// TwinCAT 3 PLC project PLC_CRIX_MOT
// Title: lcls-plc-crix-motion
// Company: SLAC
// ProjectVersion: 0.0.0
// ProgramVersion: 3.1.4023.0
// libraries:
//   LCLS General, * (SLAC)
//   lcls-twincat-motion, * (SLAC)
//   PMPS, * (SLAC - LCLS)
//   Tc2_MC2, * (Beckhoff Automation GmbH)
//   Tc2_Standard, * (Beckhoff Automation GmbH)
//   Tc2_System, * (Beckhoff Automation GmbH)
//   Tc3_EventLogger, * (Beckhoff Automation GmbH)
//   Tc3_Module, * (Beckhoff Automation GmbH)
// project tree:
//   DUTs/Assemblies/ ENUM_DiagPaddle.TcDUT (not stored), ENUM_DPX.TcDUT (not stored), ENUM_DPY.TcDUT (not stored), ENUM_DPZ.TcDUT (not stored), E_DPaddle_States.TcDUT (not stored), ST_DiagPaddleOutputs.TcDUT (not stored)
//   DUTs/EPS/ ST_BFSAssemblyState.TcDUT (not stored), ST_EPSLimits.TcDUT, ST_Queue.TcDUT (not stored)
//   GVLs/ GVL.TcGVL (not stored), GVL_DiagnosticPaddle.TcGVL (not stored), GVL_FiberLite.TcGVL, GVL_Illumination.TcGVL (not stored), GVL_MotorEPS.TcGVL, GVL_PMPS.TcGVL (not stored), GVL_PointDetector.TcGVL (not stored), GVL_Questar.TcGVL (not stored), GVL_SampleDelivery.TcGVL (not stored), Main.TcGVL
//   / PlcTask.TcTTO (not stored)
//   POUs/Assemblies/ FB_DPX.TcPOU (not stored), PRG_FZP.TcPOU, PRG_Camera.TcPOU (not stored), PRG_CryoPump.TcPOU, PRG_Cryopumps.TcPOU (not stored), PRG_CryoStat.TcPOU (not stored), PRG_DiagnosticPaddle.TcPOU (not stored), PRG_DiagnosticPaddleMotors.TcPOU (not stored), PRG_FiberLite.TcPOU, PRG_Illumination.TcPOU (not stored), PRG_InjectorMotors.TcPOU, PRG_PointDetectorMotors.TcPOU (not stored), PRG_ObjectivesMotors.TcPOU (not stored), PRG_QuestarMotors.TcPOU (not stored), PRG_RCC.TcPOU (not stored), PRG_RCI.TcPOU (not stored), PRG_VLS.TcPOU, PRG_SL2K2_SCATTER.TcPOU (not stored)
//   POUs/EPS/ FB_AdjacentStates.TcPOU (not stored), FB_AssemblyPositionStateManager.TcPOU (not stored), FB_BFS.TcPOU (not stored), FB_Queue.TcPOU (not stored), PRG_BFS.TcPOU (not stored), PRG_QueueTest.TcPOU (not stored), PRG_Test_AdjacentStates.TcPOU (not stored)
//   POUs/EPS/InjectorMotorEPSLimits/ FB_CheckEPS.TcPOU, F_InRange.TcPOU, FB_RestTimer.TcPOU, PRG_DPL_X_EPS.TcPOU, PRG_DPL_Y_EPS.TcPOU, PRG_DPL_Z_EPS.TcPOU, PRG_EPS.TcPOU, PRG_OBJ_X_EPS.TcPOU, PRG_RCC_Y_EPS.TcPOU, PRG_RCC_Z_EPS.TcPOU, PRG_SDS_RX_EPS.TcPOU, PRG_SDS_Y_EPS.TcPOU, PRG_SDS_ZENCODER_EPS.TcPOU
//   POUs/ FB_RCI_Analog_Input.TcPOU (not stored), FB_RCI_Analog_Output.TcPOU (not stored), PRG_Main.TcPOU, PRG_PMPS.TcPOU (not stored)
//   POUs/temp/ FB_SLITS.TcPOU (not stored), FB_SLITS_POWER.TcPOU (not stored), FB_SLITS_SCATTER.TcPOU (not stored)
// real-time tasks:
//   TASK PlcTask: cycle T#10ms, priority 20, ADS port 350
// motion (NC):
//   TASK NC-Task 1 SAF: cycle T#2ms, priority 4, ADS port 501
//   TASK NC-Task 1 SVB: cycle T#10ms, priority 8, ADS port 511
//   AXIS Cryo X (id 22)
//     Dynamic: AccelerationMaximum=1, DecelerationMaximum=1, Acceleration=1, Deceleration=1
//     Velo: Maximum=1.7
//     OtherSettings: AllowMotionCmdToSlave=true
//     encoder EncType=29
//       EncPara: ScaleFactorNumerator=5e-05, Offset=-31.22, MaxCount=#xffffffff, ReferenceSystem=1
//         Inc: RefSoftSyncMask=#x0000ffff
//     drive DrvType=24
//       DrvPara: Inverse=true
//         Analog: VeloReferenz=2, ScaleFactorActTorque=0.1
//         TimeComp: TaskDelayCycles=1
//     controller CtrType=2
//       CtrPara: PriorControlFactor=1
//         PosDiffControl: Range=0.5
//         PID: PosExtKp=1, DeadBandPosition=0.1
//         Observer: BandWidth=20
//   AXIS Cryo Y (id 23)
//     Dynamic: AccelerationMaximum=1, DecelerationMaximum=1, Acceleration=1, Deceleration=1
//     Velo: Maximum=1.4
//     OtherSettings: AllowMotionCmdToSlave=true
//     encoder EncType=29
//       EncPara: ScaleFactorNumerator=5e-05, Offset=-215.0149, MaxCount=#xffffffff
//         Inc: RefSoftSyncMask=#x0000ffff
//     drive DrvType=24
//       Analog: VeloReferenz=1.667, ScaleFactorActTorque=0.1
//       TimeComp: TaskDelayCycles=1
//     controller CtrType=2
//       CtrPara: PriorControlFactor=1
//         PosDiffControl: Range=0.5
//         PID: PosExtKp=1, DeadBandPosition=0.01
//         Observer: BandWidth=20
//   AXIS Cryo Z (id 24)
//     Dynamic: AccelerationMaximum=1, DecelerationMaximum=1, Acceleration=1, Deceleration=1
//     Velo: Maximum=1.7
//     OtherSettings: AllowMotionCmdToSlave=true
//     encoder EncType=29
//       EncPara: ScaleFactorNumerator=5e-05, Offset=-922337203685459, Inverse=true, MaxCount=#xffffffff, ReferenceSystem=1
//         Inc: RefSoftSyncMask=#x0000ffff
//     drive DrvType=24
//       DrvPara: Inverse=true
//         Analog: VeloReferenz=2, ScaleFactorActTorque=0.1
//         TimeComp: TaskDelayCycles=1
//     controller CtrType=2
//       CtrPara: PriorControlFactor=1
//         PosDiffControl: Range=0.5
//         PID: PosExtKp=1, DeadBandPosition=0.1
//         Observer: BandWidth=20
//   AXIS Cryo rY (id 25)
//   AXIS RCI X (id 26)
//     Dynamic: AccelerationMaximum=10, DecelerationMaximum=10, Acceleration=2, Deceleration=2
//     Velo: Maximum=0.4
//     OtherSettings: AllowMotionCmdToSlave=true
//     encoder EncType=29
//       EncPara: ScaleFactorNumerator=5e-05, Offset=-922337203685433, Inverse=true, MaxCount=#xffffffff, ReferenceSystem=1
//         Inc: RefSoftSyncMask=#x0000ffff
//     drive DrvType=24
//       Analog: VeloReferenz=2.667, ScaleFactorActTorque=0.1
//       TimeComp: TaskDelayCycles=1
//     controller CtrType=2
//       CtrPara: PriorControlFactor=1
//         PosDiffControl: Range=0.3
//         PID: PosExtKp=1, DeadBandPosition=0.1
//         Observer: BandWidth=20
//   AXIS RCI Y (id 27)
//     Dynamic: AccelerationMaximum=10, DecelerationMaximum=10, Acceleration=2, Deceleration=2
//     Velo: Maximum=1.7
//     OtherSettings: AllowMotionCmdToSlave=true
//     encoder EncType=29
//       EncPara: ScaleFactorNumerator=5e-05, Offset=-32.4565, MaxCount=#xffffffff, ReferenceSystem=1
//         Inc: RefSoftSyncMask=#x0000ffff
//     drive DrvType=24
//       Analog: VeloReferenz=2, ScaleFactorActTorque=0.1
//       TimeComp: TaskDelayCycles=1
//     controller CtrType=2
//       CtrPara: PriorControlFactor=1
//         PosDiffControl: Range=0.3
//         PID: DeadBandPosition=0.1
//         Observer: BandWidth=20
//   AXIS RCI Z (id 28)
//     Dynamic: AccelerationMaximum=10, DecelerationMaximum=10, Acceleration=2, Deceleration=2
//     Velo: Maximum=1.7
//     OtherSettings: AllowMotionCmdToSlave=true
//     encoder EncType=29
//       EncPara: ScaleFactorNumerator=5e-05, Offset=-922337203685442, Inverse=true, MaxCount=#xffffffff, ReferenceSystem=1
//         Inc: RefSoftSyncMask=#x0000ffff
//     drive DrvType=24
//       Analog: VeloReferenz=2, ScaleFactorActTorque=0.1
//       TimeComp: TaskDelayCycles=1
//     controller CtrType=2
//       CtrPara: PriorControlFactor=1
//         PosDiffControl: Range=0.3
//         PID: DeadBandPosition=0.1
//         Observer: BandWidth=20
//   AXIS RCI RX (id 29)
//     Dynamic: AccelerationMaximum=10, DecelerationMaximum=10, Acceleration=2, Deceleration=2
//     Velo: Maximum=2
//     OtherSettings: AllowMotionCmdToSlave=true
//     encoder EncType=4
//       EncPara: ScaleFactorNumerator=0.000234375, MaxCount=#x0000ffff
//         Inc: RefSoftSyncMask=#x0000ffff
//     drive DrvType=24
//       Analog: VeloReferenz=30, ScaleFactorActTorque=0.1
//       TimeComp: TaskDelayCycles=1
//     controller CtrType=2
//       CtrPara: PriorControlFactor=1
//         PosDiffControl: Range=0.3
//         PID: DeadBandPosition=0.5
//         Observer: BandWidth=20
//   AXIS FZP Y (id 30)
//     Dynamic: AccelerationMaximum=10, DecelerationMaximum=10, Acceleration=1, Deceleration=1
//     Velo: Maximum=2
//     OtherSettings: AllowMotionCmdToSlave=true
//     encoder EncType=29
//       EncPara: ScaleFactorNumerator=0.000244, Offset=-15658.9921, MaxCount=#xffffffff
//         Inc: RefSoftSyncMask=#x0000ffff
//     drive DrvType=24
//       DrvPara: Inverse=true
//         Analog: VeloReferenz=15, ScaleFactorActTorque=0.1
//         TimeComp: TaskDelayCycles=1
//     controller CtrType=2
//       CtrPara: PriorControlFactor=1
//         PosDiffControl: Range=0.5
//         PID: DeadBandPosition=0.01
//         Observer: BandWidth=20
//   AXIS FZP X (id 31)
//     Dynamic: AccelerationMaximum=10, DecelerationMaximum=10, Acceleration=1, Deceleration=1
//     Velo: Maximum=0.5
//     OtherSettings: AllowMotionCmdToSlave=true
//     encoder EncType=29
//       EncPara: ScaleFactorNumerator=0.000244, Offset=-16005.009, MaxCount=#xffffffff, ReferenceSystem=1
//         Inc: RefSoftSyncMask=#x0000ffff
//     drive DrvType=24
//       Analog: VeloReferenz=8, ScaleFactorActTorque=0.1
//       TimeComp: TaskDelayCycles=1
//     controller CtrType=2
//       CtrPara: PriorControlFactor=1
//         PosDiffControl: Range=0.5
//         PID: PosExtKp=1, DeadBandPosition=0.01
//         Observer: BandWidth=20
//   AXIS FZP Z (id 32)
//     Dynamic: AccelerationMaximum=10, DecelerationMaximum=10, Acceleration=1, Deceleration=1
//     Velo: Maximum=2
//     PositionAreaControl: Enable=false
//     OtherSettings: AllowMotionCmdToSlave=true
//     encoder EncType=29
//       EncPara: Offset=-1.0099, MaxCount=#xffffffff
//         Inc: RefSoftSyncMask=#x0000ffff
//     drive DrvType=24
//       Analog: VeloReferenz=15, ScaleFactorActTorque=0.1
//       TimeComp: TaskDelayCycles=1
//     controller CtrType=2
//       CtrPara: PriorControlFactor=1
//         PosDiffControl: Range=0.5
//         PID: DeadBandPosition=0.01
//         Observer: BandWidth=20
//   AXIS Camera X (id 33)
//   AXIS Camera Y (id 34)
//   AXIS M37-X (id 37)
//   AXIS M38-Y (id 38)
//   AXIS M39-Z (id 39)
//   AXIS M40-VLS-Slit-Top (id 40)
//     Dynamic: AccelerationMaximum=10, DecelerationMaximum=10, Acceleration=4.49102, Deceleration=4.49102, Jerk=20.1692
//     Velo: RefSearch=0.1, RefSync=0.1, SlowManual=0.5, FastManual=1, Maximum=1
//     OtherSettings: AllowMotionCmdToSlave=true, PulseDistancePos=1, PulseDistanceNeg=1
//     encoder EncType=4
//       EncPara: ScaleFactorNumerator=3.90625e-05, MaxCount=#x0000ffff
//         SoftEndMinControl: Enable=true
//         SoftEndMaxControl: Enable=true, Range=19
//         Inc: RefSoftSyncMask=#x0000ffff
//     drive DrvType=24
//       Analog: VeloReferenz=5, ScaleFactorActTorque=0.1
//       TimeComp: TaskDelayCycles=1
//     controller CtrType=2
//       CtrPara: PriorControlFactor=1
//         PosDiffControl: Range=0.1
//         PID: DeadBandPosition=0.1
//         Observer: BandWidth=20
//   AXIS M41-VLS-Slit-Bottom (id 41)
//     Dynamic: AccelerationMaximum=10, DecelerationMaximum=10, Acceleration=4.49102, Deceleration=4.49102, Jerk=20.1692
//     Velo: RefSearch=0.1, RefSync=0.1, SlowManual=0.5, FastManual=1, Maximum=1
//     OtherSettings: AllowMotionCmdToSlave=true, PulseDistancePos=1, PulseDistanceNeg=1
//     encoder EncType=4
//       EncPara: ScaleFactorNumerator=3.90625e-05, MaxCount=#x0000ffff
//         SoftEndMinControl: Enable=true
//         SoftEndMaxControl: Enable=true, Range=24.5
//         Inc: RefSoftSyncMask=#x0000ffff
//     drive DrvType=24
//       Analog: VeloReferenz=5, ScaleFactorActTorque=0.1
//       TimeComp: TaskDelayCycles=1
//     controller CtrType=2
//       CtrPara: PriorControlFactor=1
//         PosDiffControl: Range=0.1
//         PID: DeadBandPosition=0.1
//         Observer: BandWidth=20
//   AXIS M42-VLS-Slit-Right (id 42)
//     Dynamic: AccelerationMaximum=10, DecelerationMaximum=10, Acceleration=4.49102, Deceleration=4.49102, Jerk=20.1692
//     Velo: RefSearch=0.1, RefSync=0.1, SlowManual=0.5, FastManual=1, Maximum=1
//     OtherSettings: AllowMotionCmdToSlave=true, PulseDistancePos=1, PulseDistanceNeg=1
//     encoder EncType=4
//       EncPara: ScaleFactorNumerator=3.90625e-05, MaxCount=#x0000ffff
//         SoftEndMinControl: Enable=true
//         SoftEndMaxControl: Enable=true, Range=48.1
//         Inc: RefSoftSyncMask=#x0000ffff
//     drive DrvType=24
//       Analog: VeloReferenz=5, ScaleFactorActTorque=0.1
//       TimeComp: TaskDelayCycles=1
//     controller CtrType=2
//       CtrPara: PriorControlFactor=1
//         PosDiffControl: Range=0.1
//         PID: DeadBandPosition=0.1
//         Observer: BandWidth=20
//   AXIS M43-VLS-Slit-Left (id 43)
//     Dynamic: AccelerationMaximum=10, DecelerationMaximum=10, Acceleration=4.49102, Deceleration=4.49102, Jerk=20.1692
//     Velo: RefSearch=0.1, RefSync=0.1, SlowManual=0.5, FastManual=1, Maximum=0.5
//     OtherSettings: AllowMotionCmdToSlave=true, PulseDistancePos=1, PulseDistanceNeg=1
//     encoder EncType=4
//       EncPara: ScaleFactorNumerator=3.90625e-05, MaxCount=#x0000ffff
//         SoftEndMinControl: Enable=true
//         SoftEndMaxControl: Enable=true, Range=49
//         Inc: RefSoftSyncMask=#x0000ffff
//     drive DrvType=24
//       Analog: VeloReferenz=5, ScaleFactorActTorque=0.1
//       TimeComp: TaskDelayCycles=1
//     controller CtrType=2
//       CtrPara: PriorControlFactor=1
//         PosDiffControl: Range=0.1
//         PID: DeadBandPosition=0.1
//         Observer: BandWidth=20
//   AXIS M44-VLS-Mirror-Pitch (id 44)
//     Dynamic: AccelerationMaximum=4, DecelerationMaximum=4, Acceleration=1.92472, Deceleration=1.92472, Jerk=18.5227
//     Velo: RefSearch=0.01, RefSync=0.01, SlowManual=0.05, FastManual=0.1, Maximum=0.4
//     TargetPosControl: Range=0.01, Time=3
//     OtherSettings: AllowMotionCmdToSlave=true, PulseDistancePos=0.1, PulseDistanceNeg=0.1
//     encoder EncType=4
//       EncPara: ScaleFactorNumerator=7.914e-05, ScaleFactorDenominator=4, MaxCount=#x0000ffff
//         SoftEndMinControl: Range=-0.2288
//         SoftEndMaxControl: Range=1.763
//         Inc: RefMode=2, RefSoftSyncMask=#x0000ffff
//     drive DrvType=24
//       Analog: VeloReferenz=3.175, ScaleFactorActTorque=0.1
//       TimeComp: TaskDelayCycles=1
//     controller CtrType=2
//       CtrPara: PriorControlFactor=1
//         PosDiffControl: Range=0.02
//         PID: PosKp=50, DeadBandPosition=0.0001
//         Observer: BandWidth=20
//   AXIS M45-VLS-Grating-Pitch (id 45)
//   AXIS M46-VLS-Camera-Pitch (id 46)
//   AXIS M47-VLS-Camera-Dist (id 47)
//   AXIS M48- Cryopump Y10 (id 48)
//   AXIS M49- Cryopump Y11 (id 49)
//   AXIS SL2K2-BOTTOM-M50 (id 50)
//   AXIS SL2K2-TOP-M51 (id 51)
//   AXIS SL2K2-NORTH-M52 (id 52)
//   AXIS SL2K2-SOUTH-M53 (id 53)
//   AXIS Axis 1 - Diagnostic Paddle X (id 1)
//   AXIS Axis 2 - Diagnostic Paddle Y (id 2)
//   AXIS Axis 3 - Diagnostic Paddle Z (id 3)
//   AXIS Axis 4 - Objectives X (id 4)
//     Dynamic: AccelerationMaximum=1, DecelerationMaximum=1, Acceleration=1, Deceleration=1
//     Velo: Maximum=5
//     OtherSettings: AllowMotionCmdToSlave=true
//     encoder EncType=29
//       EncPara: ScaleFactorNumerator=5e-05, Offset=-35, MaxCount=#xffffffff, ReferenceSystem=1
//         SoftEndMinControl: Enable=true, Range=-2
//         SoftEndMaxControl: Enable=true, Range=32
//         Inc: RefSoftSyncMask=#x0000ffff
//     drive DrvType=24
//       DrvPara: Inverse=true
//         Analog: VeloReferenz=10, ScaleFactorActTorque=0.1
//         TimeComp: TaskDelayCycles=1
//     controller CtrType=1
//       CtrPara: PriorControlFactor=1
//         PosDiffControl: Range=1
//         Observer: BandWidth=20
//   AXIS Axis 5 - Objectives Y (id 5)
//     Dynamic: AccelerationMaximum=1, DecelerationMaximum=1, Acceleration=1, Deceleration=1
//     Velo: Maximum=5
//     OtherSettings: AllowMotionCmdToSlave=true
//     encoder EncType=29
//       EncPara: ScaleFactorNumerator=5e-05, Offset=-214688.37, MaxCount=#xffffffff, ReferenceSystem=1
//         SoftEndMinControl: Enable=true, Range=-2
//         SoftEndMaxControl: Enable=true, Range=40
//         Inc: RefSoftSyncMask=#x0000ffff
//     drive DrvType=24
//       Analog: VeloReferenz=10, ScaleFactorActTorque=0.1
//       TimeComp: TaskDelayCycles=1
//     controller CtrType=1
//       CtrPara: PriorControlFactor=1
//         PosDiffControl: Range=1
//         Observer: BandWidth=20
//   AXIS Axis 6 - Objectives Z (id 6)
//     Dynamic: AccelerationMaximum=1, DecelerationMaximum=1, Acceleration=1, Deceleration=1
//     Velo: Maximum=5
//     OtherSettings: AllowMotionCmdToSlave=true
//     encoder EncType=29
//       EncPara: ScaleFactorNumerator=5e-05, Offset=-214714.368, MaxCount=#xffffffff, ReferenceSystem=1
//         SoftEndMinControl: Enable=true, Range=-8
//         SoftEndMaxControl: Enable=true, Range=8
//         Inc: RefSoftSyncMask=#x0000ffff
//     drive DrvType=24
//       DrvPara: Inverse=true
//         Analog: VeloReferenz=10, ScaleFactorActTorque=0.1
//         TimeComp: TaskDelayCycles=1
//     controller CtrType=1
//       CtrPara: PriorControlFactor=1
//         PosDiffControl: Range=1
//         Observer: BandWidth=20
//   AXIS Axis 7 - Point Detector Y (id 7)
//     Dynamic: AccelerationMaximum=1, DecelerationMaximum=1, Acceleration=1, Deceleration=1
//     Velo: Maximum=5
//     OtherSettings: AllowMotionCmdToSlave=true
//     encoder EncType=29
//       EncPara: ScaleFactorNumerator=5e-05, MaxCount=#xffffffff
//         SoftEndMinControl: Enable=true, Range=20
//         SoftEndMaxControl: Enable=true, Range=50
//     drive DrvType=24
//       DrvPara: Inverse=true
//         Analog: VeloReferenz=10, ScaleFactorActTorque=0.1
//         TimeComp: TaskDelayCycles=1
//     controller CtrType=1
//       CtrPara: PriorControlFactor=1
//         PosDiffControl: Range=1
//         Observer: BandWidth=20
//   AXIS Axis 8 - Point Detector Rotation (id 8)
//     General: UnitName=Degree
//     Dynamic: AccelerationMaximum=1, DecelerationMaximum=1, Acceleration=1, Deceleration=1
//     Velo: Maximum=5
//     OtherSettings: AllowMotionCmdToSlave=true
//     encoder EncType=29
//       EncPara: ScaleFactorNumerator=8.3333e-08, Offset=-115, MaxCount=#xffffffff
//         SoftEndMinControl: Range=60
//         SoftEndMaxControl: Enable=true, Range=157
//     drive DrvType=24
//       Analog: VeloReferenz=20, ScaleFactorActTorque=0.1
//       TimeComp: TaskDelayCycles=1
//     controller CtrType=1
//       CtrPara: PriorControlFactor=1
//         PosDiffControl: Range=1
//         Observer: BandWidth=20
//   AXIS Axis 9 - Illumination X (id 9)
//   AXIS Axis 10 - Illumination Y (id 10)
//   AXIS Axis 11 - Illumination Z (id 11)
//   AXIS Axis 12 - Questar X (id 12)
//   AXIS Axis 13 - Questar Y (id 13)
//   AXIS Axis 14 - SPARE 1 (id 14)
//   AXIS Axis 15 - SPARE 2 (id 15)
//   AXIS Axis 16 - SDS Injector X (id 16)
//     Dynamic: AccelerationMaximum=5, DecelerationMaximum=5, Acceleration=1, Deceleration=1
//     Velo: Maximum=1
//     OtherSettings: AllowMotionCmdToSlave=true
//     encoder EncType=4
//       EncPara: ScaleFactorNumerator=0.000293, MaxCount=#xffffffff
//         Inc: RefMode=2
//     drive DrvType=24
//       DrvPara: Inverse=true
//         Analog: VeloReferenz=1.17, ScaleFactorActTorque=0.1
//         TimeComp: TaskDelayCycles=1
//     controller CtrType=2
//       CtrPara: PriorControlFactor=1
//         PosDiffControl: Range=0.5
//         PID: PosKp=5, PosExtKp=5, DeadBandPosition=0.1
//         Observer: BandWidth=20
//   AXIS Axis 17 - SDS Injectory Y (id 17)
//     Dynamic: AccelerationMaximum=5, DecelerationMaximum=5, Acceleration=1, Deceleration=1
//     Velo: Maximum=5
//     OtherSettings: AllowMotionCmdToSlave=true
//     encoder EncType=29
//       EncPara: ScaleFactorNumerator=5e-05, MaxCount=#xffffffff, ReferenceSystem=1
//     drive DrvType=24
//       Analog: VeloReferenz=10, ScaleFactorActTorque=0.1
//       TimeComp: TaskDelayCycles=1
//     controller CtrType=2
//       CtrPara: PriorControlFactor=1
//         PosDiffControl: Range=0.5
//         PID: PosKp=5, PosExtKp=1, DeadBandPosition=0.1
//         Observer: BandWidth=20
//   AXIS Axis 18 - SDS Injector Z (id 18)
//   AXIS Axis 19 - SDS Rotation X (id 19)
//     General: UnitName=Degree
//     Dynamic: AccelerationMaximum=5, DecelerationMaximum=5, Acceleration=1, Deceleration=1, Jerk=1
//     Velo: SlowManual=0.1, FastManual=0.1, Maximum=5
//     OtherSettings: AllowMotionCmdToSlave=true
//     encoder EncType=29
//       EncPara: ScaleFactorNumerator=0.1758, MaxCount=#xffffffff
//         Inc: RefSoftSyncMask=#x0000ffff
//     drive DrvType=24
//       Analog: VeloReferenz=40, ScaleFactorActTorque=0.1
//       TimeComp: TaskDelayCycles=1
//     controller CtrType=2
//       CtrPara: PriorControlFactor=1
//         PosDiffControl: Range=0.5
//         PID: PosKp=4, PosExtKp=2
//         Observer: BandWidth=20
//   AXIS Axis 20 - SDS Jet Rotation (id 20)
//     General: UnitName=Degree
//     Dynamic: AccelerationMaximum=5, DecelerationMaximum=5, Acceleration=1, Deceleration=1, Jerk=1
//     Velo: Maximum=5
//     OtherSettings: AllowMotionCmdToSlave=true
//     encoder EncType=4
//       EncPara: ScaleFactorNumerator=0.0003125, MaxCount=#x0000ffff
//         Inc: RefMode=2, RefSoftSyncMask=#x0000ffff
//     drive DrvType=24
//       Analog: VeloReferenz=40, ScaleFactorActTorque=0.1
//       TimeComp: TaskDelayCycles=1
//     controller CtrType=1
//       CtrPara: PriorControlFactor=1
//         Observer: BandWidth=20
//   AXIS Axis 21 - Questar Focus (id 21)
//   AXIS Axis 35 - Outcoupling Lens Y (id 35)
//     Dynamic: AccelerationMaximum=1, DecelerationMaximum=1, Acceleration=1, Deceleration=1
//     Velo: Maximum=5
//     OtherSettings: AllowMotionCmdToSlave=true
//     encoder EncType=29
//       EncPara: ScaleFactorNumerator=5e-05, Offset=-214688.354, MaxCount=#xffffffff, ReferenceSystem=1
//         SoftEndMinControl: Enable=true, Range=-1
//         SoftEndMaxControl: Enable=true, Range=45
//         Inc: RefSoftSyncMask=#x0000ffff
//     drive DrvType=24
//       Analog: VeloReferenz=10, ScaleFactorActTorque=0.1
//       TimeComp: TaskDelayCycles=1
//     controller CtrType=2
//       CtrPara: PriorControlFactor=1
//         PosDiffControl: Range=2.5
//         PID: PosExtKp=1, DeadBandPosition=0.01
//         Observer: BandWidth=20
//   AXIS Axis 36 - SDS Z Encoder (id 36)
//     OtherSettings: AllowMotionCmdToSlave=true
//     encoder EncType=29
//       EncPara: ScaleFactorNumerator=5e-05, MaxCount=#xffffffff, ReferenceSystem=1
//     drive DrvType=5
//       Analog: ScaleFactorActTorque=0.1
//       TimeComp: TaskDelayCycles=1
//     controller CtrType=1
//       CtrPara: PriorControlFactor=1
//         Observer: BandWidth=20
// I/O:
//   DEVICE Device 1 (EtherCAT), AmsNetId 0.0.0.0.2.1
//     Term 5 (EK1200)
// variable links:
//   (this object) <-> Device 1 (EtherCAT)/Term 5 (EK1200)/Term 6 (EK1122-0080)/DRL02-EK0 (EK1101-0080)/DRL02-ECJ1 (EK1122)/CryoStat (EK1101)/Cryo X (EL7041)
//     Drive/Inputs/In/nState1 @bit 3 <-> STM Status/Status/Error
//     Drive/Inputs/In/nState1 @bit 5 <-> STM Status/Status/Moving negative
//     Drive/Inputs/In/nState1 @bit 4 <-> STM Status/Status/Moving positive
//     Drive/Inputs/In/nState1 @bit 1 <-> STM Status/Status/Ready
//     Drive/Inputs/In/nState1 <-> STM Status/Status/Ready to enable
//     Drive/Inputs/In/nState1 @bit 6 <-> STM Status/Status/Torque reduced
//     Drive/Inputs/In/nState1 @bit 2 <-> STM Status/Status/Warning
//     Drive/Inputs/In/nState2 @bit 3 <-> STM Status/Status/Digital input 1
//     Drive/Inputs/In/nState2 @bit 4 <-> STM Status/Status/Digital input 2
//     Drive/Inputs/In/nState2 @bit 5 <-> STM Status/Status/Sync error
//     Drive/Inputs/In/nState2 @bit 7 <-> STM Status/Status/TxPDO Toggle
//     Drive/Inputs/In/nState4 @bit 1 <-> WcState/InputToggle
//     Drive/Inputs/In/nState4 <-> WcState/WcState
//     Drive/Outputs/Out/nCtrl1 <-> STM Control/Control/Enable
//     Drive/Outputs/Out/nCtrl1 @bit 2 <-> STM Control/Control/Reduce torque
//     Drive/Outputs/Out/nCtrl1 @bit 1 <-> STM Control/Control/Reset
//     Drive/Outputs/Out/nDataOut2[0] <-> STM Velocity/Velocity
//   (this object) <-> Device 1 (EtherCAT)/Term 5 (EK1200)/Term 6 (EK1122-0080)/DRL02-EK0 (EK1101-0080)/DRL02-ECJ1 (EK1122)/CryoStat (EK1101)/Cryo X/Cryo Y Enc (EL5042)
//     Enc/Inputs/In/nComState @bit 1 <-> WcState/InputToggle
//     Enc/Inputs/In/nComState <-> WcState/WcState
//     Enc/Inputs/In/nDataIn1 <-> FB Inputs Channel 1/Position
//     Enc/Inputs/In/nDataIn1 <-> FB Inputs Channel 2/Position
//     Enc/Inputs/In/nState1 @bit 12 <-> FB Inputs Channel 1/Status/Diag
//     Enc/Inputs/In/nState1 @bit 12 <-> FB Inputs Channel 2/Status/Diag
//     Enc/Inputs/In/nState1 @bit 1 <-> FB Inputs Channel 1/Status/Error
//     Enc/Inputs/In/nState1 @bit 1 <-> FB Inputs Channel 2/Status/Error
//     Enc/Inputs/In/nState1 @bit 14 <-> FB Inputs Channel 1/Status/Input cycle counter
//     Enc/Inputs/In/nState1 @bit 14 <-> FB Inputs Channel 2/Status/Input cycle counter
//     Enc/Inputs/In/nState1 @bit 2 <-> FB Inputs Channel 1/Status/Ready
//     Enc/Inputs/In/nState1 @bit 2 <-> FB Inputs Channel 2/Status/Ready
//     Enc/Inputs/In/nState1 @bit 13 <-> FB Inputs Channel 1/Status/TxPDO State
//     Enc/Inputs/In/nState1 @bit 13 <-> FB Inputs Channel 2/Status/TxPDO State
//     Enc/Inputs/In/nState1 <-> FB Inputs Channel 1/Status/Warning
//     Enc/Inputs/In/nState1 <-> FB Inputs Channel 2/Status/Warning
//   (this object) <-> Device 1 (EtherCAT)/Term 5 (EK1200)/Term 6 (EK1122-0080)/DRL02-EK0 (EK1101-0080)/DRL02-ECJ1 (EK1122)/CryoStat (EK1101)/Cryo Y (EL7041)
//     Drive/Inputs/In/nState1 @bit 3 <-> STM Status/Status/Error
//     Drive/Inputs/In/nState1 @bit 5 <-> STM Status/Status/Moving negative
//     Drive/Inputs/In/nState1 @bit 4 <-> STM Status/Status/Moving positive
//     Drive/Inputs/In/nState1 @bit 1 <-> STM Status/Status/Ready
//     Drive/Inputs/In/nState1 <-> STM Status/Status/Ready to enable
//     Drive/Inputs/In/nState1 @bit 6 <-> STM Status/Status/Torque reduced
//     Drive/Inputs/In/nState1 @bit 2 <-> STM Status/Status/Warning
//     Drive/Inputs/In/nState2 @bit 3 <-> STM Status/Status/Digital input 1
//     Drive/Inputs/In/nState2 @bit 4 <-> STM Status/Status/Digital input 2
//     Drive/Inputs/In/nState2 @bit 5 <-> STM Status/Status/Sync error
//     Drive/Inputs/In/nState2 @bit 7 <-> STM Status/Status/TxPDO Toggle
//     Drive/Inputs/In/nState4 @bit 1 <-> WcState/InputToggle
//     Drive/Inputs/In/nState4 <-> WcState/WcState
//     Drive/Outputs/Out/nCtrl1 <-> STM Control/Control/Enable
//     Drive/Outputs/Out/nCtrl1 @bit 2 <-> STM Control/Control/Reduce torque
//     Drive/Outputs/Out/nCtrl1 @bit 1 <-> STM Control/Control/Reset
//     Drive/Outputs/Out/nDataOut2[0] <-> STM Velocity/Velocity
//   (this object) <-> Device 1 (EtherCAT)/Term 5 (EK1200)/Term 6 (EK1122-0080)/DRL02-EK0 (EK1101-0080)/DRL02-ECJ1 (EK1122)/CryoStat (EK1101)/Cryo Z (EL7041)
//     Drive/Inputs/In/nState1 @bit 3 <-> STM Status/Status/Error
//     Drive/Inputs/In/nState1 @bit 5 <-> STM Status/Status/Moving negative
//     Drive/Inputs/In/nState1 @bit 4 <-> STM Status/Status/Moving positive
//     Drive/Inputs/In/nState1 @bit 1 <-> STM Status/Status/Ready
//     Drive/Inputs/In/nState1 <-> STM Status/Status/Ready to enable
//     Drive/Inputs/In/nState1 @bit 6 <-> STM Status/Status/Torque reduced
//     Drive/Inputs/In/nState1 @bit 2 <-> STM Status/Status/Warning
//     Drive/Inputs/In/nState2 @bit 3 <-> STM Status/Status/Digital input 1
//     Drive/Inputs/In/nState2 @bit 4 <-> STM Status/Status/Digital input 2
//     Drive/Inputs/In/nState2 @bit 5 <-> STM Status/Status/Sync error
//     Drive/Inputs/In/nState2 @bit 7 <-> STM Status/Status/TxPDO Toggle
//     Drive/Inputs/In/nState4 @bit 1 <-> WcState/InputToggle
//     Drive/Inputs/In/nState4 <-> WcState/WcState
//     Drive/Outputs/Out/nCtrl1 <-> STM Control/Control/Enable
//     Drive/Outputs/Out/nCtrl1 @bit 2 <-> STM Control/Control/Reduce torque
//     Drive/Outputs/Out/nCtrl1 @bit 1 <-> STM Control/Control/Reset
//     Drive/Outputs/Out/nDataOut2[0] <-> STM Velocity/Velocity
//   (this object) <-> Device 1 (EtherCAT)/Term 5 (EK1200)/Term 6 (EK1122-0080)/DRL02-EK0 (EK1101-0080)/DRL02-ECJ1 (EK1122)/CryoStat (EK1101)/Cryo Z/Cryo rY Enc (EL5042)
//     Enc/Inputs/In/nComState @bit 1 <-> WcState/InputToggle
//     Enc/Inputs/In/nComState <-> WcState/WcState
//     Enc/Inputs/In/nDataIn1 <-> FB Inputs Channel 1/Position
//     Enc/Inputs/In/nState1 @bit 12 <-> FB Inputs Channel 1/Status/Diag
//     Enc/Inputs/In/nState1 @bit 1 <-> FB Inputs Channel 1/Status/Error
//     Enc/Inputs/In/nState1 @bit 14 <-> FB Inputs Channel 1/Status/Input cycle counter
//     Enc/Inputs/In/nState1 @bit 2 <-> FB Inputs Channel 1/Status/Ready
//     Enc/Inputs/In/nState1 @bit 13 <-> FB Inputs Channel 1/Status/TxPDO State
//     Enc/Inputs/In/nState1 <-> FB Inputs Channel 1/Status/Warning
//   (this object) <-> Device 1 (EtherCAT)/Term 5 (EK1200)/Term 6 (EK1122-0080)/DRL02-EK0 (EK1101-0080)/DRL02-ECJ0 (EK1122-0080)/Term 113 (EK1101-0080)/FZP XY Enc (EL5042)
//     Enc/Inputs/In/nComState @bit 1 <-> WcState/InputToggle
//     Enc/Inputs/In/nComState <-> WcState/WcState
//     Enc/Inputs/In/nDataIn1 <-> FB Inputs Channel 1/Position
//     Enc/Inputs/In/nDataIn1 <-> FB Inputs Channel 2/Position
//     Enc/Inputs/In/nState1 @bit 12 <-> FB Inputs Channel 1/Status/Diag
//     Enc/Inputs/In/nState1 @bit 12 <-> FB Inputs Channel 2/Status/Diag
//     Enc/Inputs/In/nState1 @bit 1 <-> FB Inputs Channel 1/Status/Error
//     Enc/Inputs/In/nState1 @bit 1 <-> FB Inputs Channel 2/Status/Error
//     Enc/Inputs/In/nState1 @bit 14 <-> FB Inputs Channel 1/Status/Input cycle counter
//     Enc/Inputs/In/nState1 @bit 14 <-> FB Inputs Channel 2/Status/Input cycle counter
//     Enc/Inputs/In/nState1 @bit 2 <-> FB Inputs Channel 1/Status/Ready
//     Enc/Inputs/In/nState1 @bit 2 <-> FB Inputs Channel 2/Status/Ready
//     Enc/Inputs/In/nState1 @bit 13 <-> FB Inputs Channel 1/Status/TxPDO State
//     Enc/Inputs/In/nState1 @bit 13 <-> FB Inputs Channel 2/Status/TxPDO State
//     Enc/Inputs/In/nState1 <-> FB Inputs Channel 1/Status/Warning
//     Enc/Inputs/In/nState1 <-> FB Inputs Channel 2/Status/Warning
//   (this object) <-> Device 1 (EtherCAT)/Term 5 (EK1200)/Term 6 (EK1122-0080)/DRL02-EK0 (EK1101-0080)/DRL02-ECJ0 (EK1122-0080)/Term 113 (EK1101-0080)/FZP Y (EL7041)
//     Drive/Inputs/In/nState1 @bit 3 <-> STM Status/Status/Error
//     Drive/Inputs/In/nState1 @bit 5 <-> STM Status/Status/Moving negative
//     Drive/Inputs/In/nState1 @bit 4 <-> STM Status/Status/Moving positive
//     Drive/Inputs/In/nState1 @bit 1 <-> STM Status/Status/Ready
//     Drive/Inputs/In/nState1 <-> STM Status/Status/Ready to enable
//     Drive/Inputs/In/nState1 @bit 6 <-> STM Status/Status/Torque reduced
//     Drive/Inputs/In/nState1 @bit 2 <-> STM Status/Status/Warning
//     Drive/Inputs/In/nState2 @bit 3 <-> STM Status/Status/Digital input 1
//     Drive/Inputs/In/nState2 @bit 4 <-> STM Status/Status/Digital input 2
//     Drive/Inputs/In/nState2 @bit 5 <-> STM Status/Status/Sync error
//     Drive/Inputs/In/nState2 @bit 7 <-> STM Status/Status/TxPDO Toggle
//     Drive/Inputs/In/nState4 @bit 1 <-> WcState/InputToggle
//     Drive/Inputs/In/nState4 <-> WcState/WcState
//     Drive/Outputs/Out/nCtrl1 <-> STM Control/Control/Enable
//     Drive/Outputs/Out/nCtrl1 @bit 2 <-> STM Control/Control/Reduce torque
//     Drive/Outputs/Out/nCtrl1 @bit 1 <-> STM Control/Control/Reset
//     Drive/Outputs/Out/nDataOut2[0] <-> STM Velocity/Velocity
//   (this object) <-> Device 1 (EtherCAT)/Term 5 (EK1200)/Term 6 (EK1122-0080)/DRL02-EK0 (EK1101-0080)/DRL02-ECJ0 (EK1122-0080)/Term 113 (EK1101-0080)/FZP X (EL7041)
//     Drive/Inputs/In/nState1 @bit 3 <-> STM Status/Status/Error
//     Drive/Inputs/In/nState1 @bit 5 <-> STM Status/Status/Moving negative
//     Drive/Inputs/In/nState1 @bit 4 <-> STM Status/Status/Moving positive
//     Drive/Inputs/In/nState1 @bit 1 <-> STM Status/Status/Ready
//     Drive/Inputs/In/nState1 <-> STM Status/Status/Ready to enable
//     Drive/Inputs/In/nState1 @bit 6 <-> STM Status/Status/Torque reduced
//     Drive/Inputs/In/nState1 @bit 2 <-> STM Status/Status/Warning
//     Drive/Inputs/In/nState2 @bit 3 <-> STM Status/Status/Digital input 1
//     Drive/Inputs/In/nState2 @bit 4 <-> STM Status/Status/Digital input 2
//     Drive/Inputs/In/nState2 @bit 5 <-> STM Status/Status/Sync error
//     Drive/Inputs/In/nState2 @bit 7 <-> STM Status/Status/TxPDO Toggle
//     Drive/Inputs/In/nState4 @bit 1 <-> WcState/InputToggle
//     Drive/Inputs/In/nState4 <-> WcState/WcState
//     Drive/Outputs/Out/nCtrl1 <-> STM Control/Control/Enable
//     Drive/Outputs/Out/nCtrl1 @bit 2 <-> STM Control/Control/Reduce torque
//     Drive/Outputs/Out/nCtrl1 @bit 1 <-> STM Control/Control/Reset
//     Drive/Outputs/Out/nDataOut2[0] <-> STM Velocity/Velocity
//   (this object) <-> Device 1 (EtherCAT)/Term 5 (EK1200)/Term 6 (EK1122-0080)/DRL02-EK0 (EK1101-0080)/DRL02-ECJ0 (EK1122-0080)/Term 113 (EK1101-0080)/FZP Z (EL7041)
//     Drive/Inputs/In/nState1 @bit 3 <-> STM Status/Status/Error
//     Drive/Inputs/In/nState1 @bit 5 <-> STM Status/Status/Moving negative
//     Drive/Inputs/In/nState1 @bit 4 <-> STM Status/Status/Moving positive
//     Drive/Inputs/In/nState1 @bit 1 <-> STM Status/Status/Ready
//     Drive/Inputs/In/nState1 <-> STM Status/Status/Ready to enable
//     Drive/Inputs/In/nState1 @bit 6 <-> STM Status/Status/Torque reduced
//     Drive/Inputs/In/nState1 @bit 2 <-> STM Status/Status/Warning
//     Drive/Inputs/In/nState2 @bit 3 <-> STM Status/Status/Digital input 1
//     Drive/Inputs/In/nState2 @bit 4 <-> STM Status/Status/Digital input 2
//     Drive/Inputs/In/nState2 @bit 5 <-> STM Status/Status/Sync error
//     Drive/Inputs/In/nState2 @bit 7 <-> STM Status/Status/TxPDO Toggle
//     Drive/Inputs/In/nState4 @bit 1 <-> WcState/InputToggle
//     Drive/Inputs/In/nState4 <-> WcState/WcState
//     Drive/Outputs/Out/nCtrl1 <-> STM Control/Control/Enable
//     Drive/Outputs/Out/nCtrl1 @bit 2 <-> STM Control/Control/Reduce torque
//     Drive/Outputs/Out/nCtrl1 @bit 1 <-> STM Control/Control/Reset
//     Drive/Outputs/Out/nDataOut2[0] <-> STM Velocity/Velocity
//   (this object) <-> Device 1 (EtherCAT)/Term 5 (EK1200)/Term 6 (EK1122-0080)/DRL02-EK0 (EK1101-0080)/DRL02-ECJ0 (EK1122-0080)/Term 113 (EK1101-0080)/FZP Z Enc (EL5042)
//     Enc/Inputs/In/nComState @bit 1 <-> WcState/InputToggle
//     Enc/Inputs/In/nComState <-> WcState/WcState
//     Enc/Inputs/In/nDataIn1 <-> FB Inputs Channel 2/Position
//     Enc/Inputs/In/nState1 @bit 12 <-> FB Inputs Channel 2/Status/Diag
//     Enc/Inputs/In/nState1 @bit 1 <-> FB Inputs Channel 2/Status/Error
//     Enc/Inputs/In/nState1 @bit 14 <-> FB Inputs Channel 2/Status/Input cycle counter
//     Enc/Inputs/In/nState1 @bit 2 <-> FB Inputs Channel 2/Status/Ready
//     Enc/Inputs/In/nState1 @bit 13 <-> FB Inputs Channel 2/Status/TxPDO State
//     Enc/Inputs/In/nState1 <-> FB Inputs Channel 2/Status/Warning
//   (this object) <-> Device 1 (EtherCAT)/Term 5 (EK1200)/Term 6 (EK1122-0080)/DRL02-EK0 (EK1101-0080)/DRL02-ECJ1 (EK1122)/VLS_EP6_EP7041-1002
//     Drive/Inputs/In/nState1 @bit 3 <-> STM Status/Status/Error
//     Drive/Inputs/In/nState1 @bit 5 <-> STM Status/Status/Moving negative
//     Drive/Inputs/In/nState1 @bit 4 <-> STM Status/Status/Moving positive
//     Drive/Inputs/In/nState1 @bit 1 <-> STM Status/Status/Ready
//     Drive/Inputs/In/nState1 <-> STM Status/Status/Ready to enable
//     Drive/Inputs/In/nState1 @bit 6 <-> STM Status/Status/Torque reduced
//     Drive/Inputs/In/nState1 @bit 2 <-> STM Status/Status/Warning
//     Drive/Inputs/In/nState2 @bit 3 <-> STM Status/Status/Digital input 1
//     Drive/Inputs/In/nState2 @bit 4 <-> STM Status/Status/Digital input 2
//     Drive/Inputs/In/nState2 @bit 5 <-> STM Status/Status/Sync error
//     Drive/Inputs/In/nState2 @bit 7 <-> STM Status/Status/TxPDO Toggle
//     Drive/Inputs/In/nState4 @bit 1 <-> WcState/InputToggle
//     Drive/Inputs/In/nState4 <-> WcState/WcState
//     Drive/Outputs/Out/nCtrl1 <-> STM Control/Control/Enable
//     Drive/Outputs/Out/nCtrl1 @bit 2 <-> STM Control/Control/Reduce torque
//     Drive/Outputs/Out/nCtrl1 @bit 1 <-> STM Control/Control/Reset
//     Drive/Outputs/Out/nCtrl2 @bit 3 <-> STM Control/Control/Digital output 1
//     Drive/Outputs/Out/nDataOut2[0] <-> STM Velocity/Velocity
//     Enc/Inputs/In/nDataIn1[0] <-> ENC Status compact/Counter value
//     Enc/Inputs/In/nDataIn2[0] <-> ENC Status compact/Latch value
//     Enc/Inputs/In/nState1 @bit 4 <-> ENC Status compact/Status/Counter overflow
//     Enc/Inputs/In/nState1 @bit 3 <-> ENC Status compact/Status/Counter underflow
//     Enc/Inputs/In/nState1 @bit 7 <-> ENC Status compact/Status/Extrapolation stall
//     Enc/Inputs/In/nState1 <-> ENC Status compact/Status/Latch C valid
//     Enc/Inputs/In/nState1 @bit 1 <-> ENC Status compact/Status/Latch extern valid
//     Enc/Inputs/In/nState1 @bit 2 <-> ENC Status compact/Status/Set counter done
//     Enc/Inputs/In/nState2 @bit 4 <-> ENC Status compact/Status/Status of extern latch
//     Enc/Inputs/In/nState2 <-> ENC Status compact/Status/Status of input A
//     Enc/Inputs/In/nState2 @bit 1 <-> ENC Status compact/Status/Status of input B
//     Enc/Inputs/In/nState2 @bit 2 <-> ENC Status compact/Status/Status of input C
//     Enc/Inputs/In/nState2 @bit 5 <-> ENC Status compact/Status/Sync error
//     Enc/Inputs/In/nState2 @bit 7 <-> ENC Status compact/Status/TxPDO Toggle
//     Enc/Inputs/In/nState4 @bit 1 <-> WcState/InputToggle
//     Enc/Inputs/In/nState4 <-> WcState/WcState
//     Enc/Outputs/Out/nCtrl1 <-> ENC Control compact/Control/Enable latch C
//     Enc/Outputs/Out/nCtrl1 @bit 3 <-> ENC Control compact/Control/Enable latch extern on negative edge
//     Enc/Outputs/Out/nCtrl1 @bit 1 <-> ENC Control compact/Control/Enable latch extern on positive edge
//     Enc/Outputs/Out/nCtrl1 @bit 2 <-> ENC Control compact/Control/Set counter
//     Enc/Outputs/Out/nDataOut1[0] <-> ENC Control compact/Set counter value
//   (this object) <-> Device 1 (EtherCAT)/Term 5 (EK1200)/Term 6 (EK1122-0080)/DRL02-EK0 (EK1101-0080)/DRL02-ECJ1 (EK1122)/VLS_EP7_EP7041-1002
//     Drive/Inputs/In/nState1 @bit 3 <-> STM Status/Status/Error
//     Drive/Inputs/In/nState1 @bit 5 <-> STM Status/Status/Moving negative
//     Drive/Inputs/In/nState1 @bit 4 <-> STM Status/Status/Moving positive
//     Drive/Inputs/In/nState1 @bit 1 <-> STM Status/Status/Ready
//     Drive/Inputs/In/nState1 <-> STM Status/Status/Ready to enable
//     Drive/Inputs/In/nState1 @bit 6 <-> STM Status/Status/Torque reduced
//     Drive/Inputs/In/nState1 @bit 2 <-> STM Status/Status/Warning
//     Drive/Inputs/In/nState2 @bit 3 <-> STM Status/Status/Digital input 1
//     Drive/Inputs/In/nState2 @bit 4 <-> STM Status/Status/Digital input 2
//     Drive/Inputs/In/nState2 @bit 5 <-> STM Status/Status/Sync error
//     Drive/Inputs/In/nState2 @bit 7 <-> STM Status/Status/TxPDO Toggle
//     Drive/Inputs/In/nState4 @bit 1 <-> WcState/InputToggle
//     Drive/Inputs/In/nState4 <-> WcState/WcState
//     Drive/Outputs/Out/nCtrl1 <-> STM Control/Control/Enable
//     Drive/Outputs/Out/nCtrl1 @bit 2 <-> STM Control/Control/Reduce torque
//     Drive/Outputs/Out/nCtrl1 @bit 1 <-> STM Control/Control/Reset
//     Drive/Outputs/Out/nCtrl2 @bit 3 <-> STM Control/Control/Digital output 1
//     Drive/Outputs/Out/nDataOut2[0] <-> STM Velocity/Velocity
//     Enc/Inputs/In/nDataIn1[0] <-> ENC Status compact/Counter value
//     Enc/Inputs/In/nDataIn2[0] <-> ENC Status compact/Latch value
//     Enc/Inputs/In/nState1 @bit 4 <-> ENC Status compact/Status/Counter overflow
//     Enc/Inputs/In/nState1 @bit 3 <-> ENC Status compact/Status/Counter underflow
//     Enc/Inputs/In/nState1 @bit 7 <-> ENC Status compact/Status/Extrapolation stall
//     Enc/Inputs/In/nState1 <-> ENC Status compact/Status/Latch C valid
//     Enc/Inputs/In/nState1 @bit 1 <-> ENC Status compact/Status/Latch extern valid
//     Enc/Inputs/In/nState1 @bit 2 <-> ENC Status compact/Status/Set counter done
//     Enc/Inputs/In/nState2 @bit 4 <-> ENC Status compact/Status/Status of extern latch
//     Enc/Inputs/In/nState2 <-> ENC Status compact/Status/Status of input A
//     Enc/Inputs/In/nState2 @bit 1 <-> ENC Status compact/Status/Status of input B
//     Enc/Inputs/In/nState2 @bit 2 <-> ENC Status compact/Status/Status of input C
//     Enc/Inputs/In/nState2 @bit 5 <-> ENC Status compact/Status/Sync error
//     Enc/Inputs/In/nState2 @bit 7 <-> ENC Status compact/Status/TxPDO Toggle
//     Enc/Inputs/In/nState4 @bit 1 <-> WcState/InputToggle
//     Enc/Inputs/In/nState4 <-> WcState/WcState
//     Enc/Outputs/Out/nCtrl1 <-> ENC Control compact/Control/Enable latch C
//     Enc/Outputs/Out/nCtrl1 @bit 3 <-> ENC Control compact/Control/Enable latch extern on negative edge
//     Enc/Outputs/Out/nCtrl1 @bit 1 <-> ENC Control compact/Control/Enable latch extern on positive edge
//     Enc/Outputs/Out/nCtrl1 @bit 2 <-> ENC Control compact/Control/Set counter
//     Enc/Outputs/Out/nDataOut1[0] <-> ENC Control compact/Set counter value
//   (this object) <-> Device 1 (EtherCAT)/Term 5 (EK1200)/Term 6 (EK1122-0080)/DRL02-EK0 (EK1101-0080)/DRL02-ECJ1 (EK1122)/VLS_EP8_EP7041-1002
//     Drive/Inputs/In/nState1 @bit 3 <-> STM Status/Status/Error
//     Drive/Inputs/In/nState1 @bit 5 <-> STM Status/Status/Moving negative
//     Drive/Inputs/In/nState1 @bit 4 <-> STM Status/Status/Moving positive
//     Drive/Inputs/In/nState1 @bit 1 <-> STM Status/Status/Ready
//     Drive/Inputs/In/nState1 <-> STM Status/Status/Ready to enable
//     Drive/Inputs/In/nState1 @bit 6 <-> STM Status/Status/Torque reduced
//     Drive/Inputs/In/nState1 @bit 2 <-> STM Status/Status/Warning
//     Drive/Inputs/In/nState2 @bit 3 <-> STM Status/Status/Digital input 1
//     Drive/Inputs/In/nState2 @bit 4 <-> STM Status/Status/Digital input 2
//     Drive/Inputs/In/nState2 @bit 5 <-> STM Status/Status/Sync error
//     Drive/Inputs/In/nState2 @bit 7 <-> STM Status/Status/TxPDO Toggle
//     Drive/Inputs/In/nState4 @bit 1 <-> WcState/InputToggle
//     Drive/Inputs/In/nState4 <-> WcState/WcState
//     Drive/Outputs/Out/nCtrl1 <-> STM Control/Control/Enable
//     Drive/Outputs/Out/nCtrl1 @bit 2 <-> STM Control/Control/Reduce torque
//     Drive/Outputs/Out/nCtrl1 @bit 1 <-> STM Control/Control/Reset
//     Drive/Outputs/Out/nCtrl2 @bit 3 <-> STM Control/Control/Digital output 1
//     Drive/Outputs/Out/nDataOut2[0] <-> STM Velocity/Velocity
//     Enc/Inputs/In/nDataIn1[0] <-> ENC Status compact/Counter value
//     Enc/Inputs/In/nDataIn2[0] <-> ENC Status compact/Latch value
//     Enc/Inputs/In/nState1 @bit 4 <-> ENC Status compact/Status/Counter overflow
//     Enc/Inputs/In/nState1 @bit 3 <-> ENC Status compact/Status/Counter underflow
//     Enc/Inputs/In/nState1 @bit 7 <-> ENC Status compact/Status/Extrapolation stall
//     Enc/Inputs/In/nState1 <-> ENC Status compact/Status/Latch C valid
//     Enc/Inputs/In/nState1 @bit 1 <-> ENC Status compact/Status/Latch extern valid
//     Enc/Inputs/In/nState1 @bit 2 <-> ENC Status compact/Status/Set counter done
//     Enc/Inputs/In/nState2 @bit 4 <-> ENC Status compact/Status/Status of extern latch
//     Enc/Inputs/In/nState2 <-> ENC Status compact/Status/Status of input A
//     Enc/Inputs/In/nState2 @bit 1 <-> ENC Status compact/Status/Status of input B
//     Enc/Inputs/In/nState2 @bit 2 <-> ENC Status compact/Status/Status of input C
//     Enc/Inputs/In/nState2 @bit 5 <-> ENC Status compact/Status/Sync error
//     Enc/Inputs/In/nState2 @bit 7 <-> ENC Status compact/Status/TxPDO Toggle
//     Enc/Inputs/In/nState4 @bit 1 <-> WcState/InputToggle
//     Enc/Inputs/In/nState4 <-> WcState/WcState
//     Enc/Outputs/Out/nCtrl1 <-> ENC Control compact/Control/Enable latch C
//     Enc/Outputs/Out/nCtrl1 @bit 3 <-> ENC Control compact/Control/Enable latch extern on negative edge
//     Enc/Outputs/Out/nCtrl1 @bit 1 <-> ENC Control compact/Control/Enable latch extern on positive edge
//     Enc/Outputs/Out/nCtrl1 @bit 2 <-> ENC Control compact/Control/Set counter
//     Enc/Outputs/Out/nDataOut1[0] <-> ENC Control compact/Set counter value
//   (this object) <-> Device 1 (EtherCAT)/Term 5 (EK1200)/Term 6 (EK1122-0080)/DRL02-EK0 (EK1101-0080)/DRL02-ECJ1 (EK1122)/VLS_EP9_EP7041-1002
//     Drive/Inputs/In/nState1 @bit 3 <-> STM Status/Status/Error
//     Drive/Inputs/In/nState1 @bit 5 <-> STM Status/Status/Moving negative
//     Drive/Inputs/In/nState1 @bit 4 <-> STM Status/Status/Moving positive
//     Drive/Inputs/In/nState1 @bit 1 <-> STM Status/Status/Ready
//     Drive/Inputs/In/nState1 <-> STM Status/Status/Ready to enable
//     Drive/Inputs/In/nState1 @bit 6 <-> STM Status/Status/Torque reduced
//     Drive/Inputs/In/nState1 @bit 2 <-> STM Status/Status/Warning
//     Drive/Inputs/In/nState2 @bit 3 <-> STM Status/Status/Digital input 1
//     Drive/Inputs/In/nState2 @bit 4 <-> STM Status/Status/Digital input 2
//     Drive/Inputs/In/nState2 @bit 5 <-> STM Status/Status/Sync error
//     Drive/Inputs/In/nState2 @bit 7 <-> STM Status/Status/TxPDO Toggle
//     Drive/Inputs/In/nState4 @bit 1 <-> WcState/InputToggle
//     Drive/Inputs/In/nState4 <-> WcState/WcState
//     Drive/Outputs/Out/nCtrl1 <-> STM Control/Control/Enable
//     Drive/Outputs/Out/nCtrl1 @bit 2 <-> STM Control/Control/Reduce torque
//     Drive/Outputs/Out/nCtrl1 @bit 1 <-> STM Control/Control/Reset
//     Drive/Outputs/Out/nCtrl2 @bit 3 <-> STM Control/Control/Digital output 1
//     Drive/Outputs/Out/nDataOut2[0] <-> STM Velocity/Velocity
//     Enc/Inputs/In/nDataIn1[0] <-> ENC Status compact/Counter value
//     Enc/Inputs/In/nDataIn2[0] <-> ENC Status compact/Latch value
//     Enc/Inputs/In/nState1 @bit 4 <-> ENC Status compact/Status/Counter overflow
//     Enc/Inputs/In/nState1 @bit 3 <-> ENC Status compact/Status/Counter underflow
//     Enc/Inputs/In/nState1 @bit 7 <-> ENC Status compact/Status/Extrapolation stall
//     Enc/Inputs/In/nState1 <-> ENC Status compact/Status/Latch C valid
//     Enc/Inputs/In/nState1 @bit 1 <-> ENC Status compact/Status/Latch extern valid
//     Enc/Inputs/In/nState1 @bit 2 <-> ENC Status compact/Status/Set counter done
//     Enc/Inputs/In/nState2 @bit 4 <-> ENC Status compact/Status/Status of extern latch
//     Enc/Inputs/In/nState2 <-> ENC Status compact/Status/Status of input A
//     Enc/Inputs/In/nState2 @bit 1 <-> ENC Status compact/Status/Status of input B
//     Enc/Inputs/In/nState2 @bit 2 <-> ENC Status compact/Status/Status of input C
//     Enc/Inputs/In/nState2 @bit 5 <-> ENC Status compact/Status/Sync error
//     Enc/Inputs/In/nState2 @bit 7 <-> ENC Status compact/Status/TxPDO Toggle
//     Enc/Inputs/In/nState4 @bit 1 <-> WcState/InputToggle
//     Enc/Inputs/In/nState4 <-> WcState/WcState
//     Enc/Outputs/Out/nCtrl1 <-> ENC Control compact/Control/Enable latch C
//     Enc/Outputs/Out/nCtrl1 @bit 3 <-> ENC Control compact/Control/Enable latch extern on negative edge
//     Enc/Outputs/Out/nCtrl1 @bit 1 <-> ENC Control compact/Control/Enable latch extern on positive edge
//     Enc/Outputs/Out/nCtrl1 @bit 2 <-> ENC Control compact/Control/Set counter
//     Enc/Outputs/Out/nDataOut1[0] <-> ENC Control compact/Set counter value
//   (this object) <-> Device 1 (EtherCAT)/Term 5 (EK1200)/Term 6 (EK1122-0080)/DRL02-EK0 (EK1101-0080)/DRL02-ECJ1 (EK1122)/VLS_EP10_EP7041-3102
//     Drive/Inputs/In/nState1 @bit 3 <-> STM Status/Status/Error
//     Drive/Inputs/In/nState1 @bit 7 <-> STM Status/Status/Motor stall
//     Drive/Inputs/In/nState1 @bit 5 <-> STM Status/Status/Moving negative
//     Drive/Inputs/In/nState1 @bit 4 <-> STM Status/Status/Moving positive
//     Drive/Inputs/In/nState1 @bit 1 <-> STM Status/Status/Ready
//     Drive/Inputs/In/nState1 <-> STM Status/Status/Ready to enable
//     Drive/Inputs/In/nState1 @bit 6 <-> STM Status/Status/Torque reduced
//     Drive/Inputs/In/nState1 @bit 2 <-> STM Status/Status/Warning
//     Drive/Inputs/In/nState2 @bit 3 <-> STM Status/Status/Digital input 1
//     Drive/Inputs/In/nState2 @bit 4 <-> STM Status/Status/Digital input 2
//     Drive/Inputs/In/nState2 @bit 5 <-> STM Status/Status/Sync error
//     Drive/Inputs/In/nState2 @bit 7 <-> STM Status/Status/TxPDO Toggle
//     Drive/Inputs/In/nState4 @bit 1 <-> WcState/InputToggle
//     Drive/Inputs/In/nState4 <-> WcState/WcState
//     Drive/Outputs/Out/nCtrl1 <-> STM Control/Control/Enable
//     Drive/Outputs/Out/nCtrl1 @bit 2 <-> STM Control/Control/Reduce torque
//     Drive/Outputs/Out/nCtrl1 @bit 1 <-> STM Control/Control/Reset
//     Drive/Outputs/Out/nCtrl2 @bit 3 <-> STM Control/Control/Digital output 1
//     Drive/Outputs/Out/nDataOut2[0] <-> STM Velocity/Velocity
//     Enc/Inputs/In/nDataIn1[0] <-> ENC Status compact/Counter value
//     Enc/Inputs/In/nDataIn2[0] <-> ENC Status compact/Latch value
//     Enc/Inputs/In/nState1 @bit 4 <-> ENC Status compact/Status/Counter overflow
//     Enc/Inputs/In/nState1 @bit 3 <-> ENC Status compact/Status/Counter underflow
//     Enc/Inputs/In/nState1 @bit 7 <-> ENC Status compact/Status/Extrapolation stall
//     Enc/Inputs/In/nState1 <-> ENC Status compact/Status/Latch C valid
//     Enc/Inputs/In/nState1 @bit 1 <-> ENC Status compact/Status/Latch extern valid
//     Enc/Inputs/In/nState1 @bit 2 <-> ENC Status compact/Status/Set counter done
//     Enc/Inputs/In/nState2 @bit 4 <-> ENC Status compact/Status/Status of extern latch
//     Enc/Inputs/In/nState2 <-> ENC Status compact/Status/Status of input A
//     Enc/Inputs/In/nState2 @bit 1 <-> ENC Status compact/Status/Status of input B
//     Enc/Inputs/In/nState2 @bit 2 <-> ENC Status compact/Status/Status of input C
//     Enc/Inputs/In/nState2 @bit 5 <-> ENC Status compact/Status/Sync error
//     Enc/Inputs/In/nState2 @bit 7 <-> ENC Status compact/Status/TxPDO Toggle
//     Enc/Inputs/In/nState4 @bit 1 <-> WcState/InputToggle
//     Enc/Inputs/In/nState4 <-> WcState/WcState
//     Enc/Outputs/Out/nCtrl1 <-> ENC Control compact/Control/Enable latch C
//     Enc/Outputs/Out/nCtrl1 @bit 3 <-> ENC Control compact/Control/Enable latch extern on negative edge
//     Enc/Outputs/Out/nCtrl1 @bit 1 <-> ENC Control compact/Control/Enable latch extern on positive edge
//     Enc/Outputs/Out/nCtrl1 @bit 2 <-> ENC Control compact/Control/Set counter
//     Enc/Outputs/Out/nDataOut1[0] <-> ENC Control compact/Set counter value
//   (this object) <-> Device 1 (EtherCAT)/Term 5 (EK1200)/Term 6 (EK1122-0080)/DRL02-EK0 (EK1101-0080)/DRL02-E5 (EL5042)
//     Enc/Inputs/In/nComState @bit 1 <-> WcState/InputToggle
//     Enc/Inputs/In/nComState <-> WcState/WcState
//     Enc/Inputs/In/nDataIn1 <-> FB Inputs Channel 2/Position
//     Enc/Inputs/In/nState1 @bit 12 <-> FB Inputs Channel 2/Status/Diag
//     Enc/Inputs/In/nState1 @bit 1 <-> FB Inputs Channel 2/Status/Error
//     Enc/Inputs/In/nState1 @bit 14 <-> FB Inputs Channel 2/Status/Input cycle counter
//     Enc/Inputs/In/nState1 @bit 2 <-> FB Inputs Channel 2/Status/Ready
//     Enc/Inputs/In/nState1 @bit 13 <-> FB Inputs Channel 2/Status/TxPDO State
//     Enc/Inputs/In/nState1 <-> FB Inputs Channel 2/Status/Warning
//   (this object) <-> Device 1 (EtherCAT)/Term 5 (EK1200)/Term 6 (EK1122-0080)/DRL02-EK0 (EK1101-0080)/DRL02-E6 (EL7031)
//     Drive/Inputs/In/nState1 @bit 3 <-> STM Status/Status/Error
//     Drive/Inputs/In/nState1 @bit 5 <-> STM Status/Status/Moving negative
//     Drive/Inputs/In/nState1 @bit 4 <-> STM Status/Status/Moving positive
//     Drive/Inputs/In/nState1 @bit 1 <-> STM Status/Status/Ready
//     Drive/Inputs/In/nState1 <-> STM Status/Status/Ready to enable
//     Drive/Inputs/In/nState1 @bit 6 <-> STM Status/Status/Torque reduced
//     Drive/Inputs/In/nState1 @bit 2 <-> STM Status/Status/Warning
//     Drive/Inputs/In/nState2 @bit 3 <-> STM Status/Status/Digital input 1
//     Drive/Inputs/In/nState2 @bit 4 <-> STM Status/Status/Digital input 2
//     Drive/Inputs/In/nState2 @bit 5 <-> STM Status/Status/Sync error
//     Drive/Inputs/In/nState2 @bit 7 <-> STM Status/Status/TxPDO Toggle
//     Drive/Inputs/In/nState4 @bit 1 <-> WcState/InputToggle
//     Drive/Inputs/In/nState4 <-> WcState/WcState
//     Drive/Outputs/Out/nCtrl1 <-> STM Control/Control/Enable
//     Drive/Outputs/Out/nCtrl1 @bit 2 <-> STM Control/Control/Reduce torque
//     Drive/Outputs/Out/nCtrl1 @bit 1 <-> STM Control/Control/Reset
//     Drive/Outputs/Out/nDataOut2[0] <-> STM Velocity/Velocity
//   (this object) <-> Device 1 (EtherCAT)/Term 5 (EK1200)/Term 6 (EK1122-0080)/DRL02-EK0 (EK1101-0080)/DRL02-E7 (EL7031)
//     Drive/Inputs/In/nState1 @bit 3 <-> STM Status/Status/Error
//     Drive/Inputs/In/nState1 @bit 5 <-> STM Status/Status/Moving negative
//     Drive/Inputs/In/nState1 @bit 4 <-> STM Status/Status/Moving positive
//     Drive/Inputs/In/nState1 @bit 1 <-> STM Status/Status/Ready
//     Drive/Inputs/In/nState1 <-> STM Status/Status/Ready to enable
//     Drive/Inputs/In/nState1 @bit 6 <-> STM Status/Status/Torque reduced
//     Drive/Inputs/In/nState1 @bit 2 <-> STM Status/Status/Warning
//     Drive/Inputs/In/nState2 @bit 3 <-> STM Status/Status/Digital input 1
//     Drive/Inputs/In/nState2 @bit 4 <-> STM Status/Status/Digital input 2
//     Drive/Inputs/In/nState2 @bit 5 <-> STM Status/Status/Sync error
//     Drive/Inputs/In/nState2 @bit 7 <-> STM Status/Status/TxPDO Toggle
//     Drive/Inputs/In/nState4 @bit 1 <-> WcState/InputToggle
//     Drive/Inputs/In/nState4 <-> WcState/WcState
//     Drive/Outputs/Out/nCtrl1 <-> STM Control/Control/Enable
//     Drive/Outputs/Out/nCtrl1 @bit 2 <-> STM Control/Control/Reduce torque
//     Drive/Outputs/Out/nCtrl1 @bit 1 <-> STM Control/Control/Reset
//     Drive/Outputs/Out/nDataOut2[0] <-> STM Velocity/Velocity
//   (this object) <-> Device 1 (EtherCAT)/Term 5 (EK1200)/Term 6 (EK1122-0080)/DRL02-EK0 (EK1101-0080)/DRL02-E8 (EL5042)
//     Enc/Inputs/In/nComState @bit 1 <-> WcState/InputToggle
//     Enc/Inputs/In/nComState <-> WcState/WcState
//     Enc/Inputs/In/nDataIn1 <-> FB Inputs Channel 1/Position
//     Enc/Inputs/In/nDataIn1 <-> FB Inputs Channel 2/Position
//     Enc/Inputs/In/nState1 @bit 12 <-> FB Inputs Channel 1/Status/Diag
//     Enc/Inputs/In/nState1 @bit 12 <-> FB Inputs Channel 2/Status/Diag
//     Enc/Inputs/In/nState1 @bit 1 <-> FB Inputs Channel 1/Status/Error
//     Enc/Inputs/In/nState1 @bit 1 <-> FB Inputs Channel 2/Status/Error
//     Enc/Inputs/In/nState1 @bit 14 <-> FB Inputs Channel 1/Status/Input cycle counter
//     Enc/Inputs/In/nState1 @bit 14 <-> FB Inputs Channel 2/Status/Input cycle counter
//     Enc/Inputs/In/nState1 @bit 2 <-> FB Inputs Channel 1/Status/Ready
//     Enc/Inputs/In/nState1 @bit 2 <-> FB Inputs Channel 2/Status/Ready
//     Enc/Inputs/In/nState1 @bit 13 <-> FB Inputs Channel 1/Status/TxPDO State
//     Enc/Inputs/In/nState1 @bit 13 <-> FB Inputs Channel 2/Status/TxPDO State
//     Enc/Inputs/In/nState1 <-> FB Inputs Channel 1/Status/Warning
//     Enc/Inputs/In/nState1 <-> FB Inputs Channel 2/Status/Warning
//   (this object) <-> Device 1 (EtherCAT)/Term 5 (EK1200)/Term 6 (EK1122-0080)/DRL02-EK0 (EK1101-0080)/DRL02-E9 (EL7031)
//     Drive/Inputs/In/nState1 @bit 3 <-> STM Status/Status/Error
//     Drive/Inputs/In/nState1 @bit 5 <-> STM Status/Status/Moving negative
//     Drive/Inputs/In/nState1 @bit 4 <-> STM Status/Status/Moving positive
//     Drive/Inputs/In/nState1 @bit 1 <-> STM Status/Status/Ready
//     Drive/Inputs/In/nState1 <-> STM Status/Status/Ready to enable
//     Drive/Inputs/In/nState1 @bit 6 <-> STM Status/Status/Torque reduced
//     Drive/Inputs/In/nState1 @bit 2 <-> STM Status/Status/Warning
//     Drive/Inputs/In/nState2 @bit 3 <-> STM Status/Status/Digital input 1
//     Drive/Inputs/In/nState2 @bit 4 <-> STM Status/Status/Digital input 2
//     Drive/Inputs/In/nState2 @bit 5 <-> STM Status/Status/Sync error
//     Drive/Inputs/In/nState2 @bit 7 <-> STM Status/Status/TxPDO Toggle
//     Drive/Inputs/In/nState4 @bit 1 <-> WcState/InputToggle
//     Drive/Inputs/In/nState4 <-> WcState/WcState
//     Drive/Outputs/Out/nCtrl1 <-> STM Control/Control/Enable
//     Drive/Outputs/Out/nCtrl1 @bit 2 <-> STM Control/Control/Reduce torque
//     Drive/Outputs/Out/nCtrl1 @bit 1 <-> STM Control/Control/Reset
//     Drive/Outputs/Out/nDataOut2[0] <-> STM Velocity/Velocity
//   (this object) <-> Device 1 (EtherCAT)/Term 5 (EK1200)/Term 6 (EK1122-0080)/DRL02-EK0 (EK1101-0080)/DRL02-E11 (EL7031)
//     Drive/Inputs/In/nState1 @bit 3 <-> STM Status/Status/Error
//     Drive/Inputs/In/nState1 @bit 5 <-> STM Status/Status/Moving negative
//     Drive/Inputs/In/nState1 @bit 4 <-> STM Status/Status/Moving positive
//     Drive/Inputs/In/nState1 @bit 1 <-> STM Status/Status/Ready
//     Drive/Inputs/In/nState1 <-> STM Status/Status/Ready to enable
//     Drive/Inputs/In/nState1 @bit 6 <-> STM Status/Status/Torque reduced
//     Drive/Inputs/In/nState1 @bit 2 <-> STM Status/Status/Warning
//     Drive/Inputs/In/nState2 @bit 3 <-> STM Status/Status/Digital input 1
//     Drive/Inputs/In/nState2 @bit 4 <-> STM Status/Status/Digital input 2
//     Drive/Inputs/In/nState2 @bit 5 <-> STM Status/Status/Sync error
//     Drive/Inputs/In/nState2 @bit 7 <-> STM Status/Status/TxPDO Toggle
//     Drive/Inputs/In/nState4 @bit 1 <-> WcState/InputToggle
//     Drive/Inputs/In/nState4 <-> WcState/WcState
//     Drive/Outputs/Out/nCtrl1 <-> STM Control/Control/Enable
//     Drive/Outputs/Out/nCtrl1 @bit 2 <-> STM Control/Control/Reduce torque
//     Drive/Outputs/Out/nCtrl1 @bit 1 <-> STM Control/Control/Reset
//     Drive/Outputs/Out/nDataOut2[0] <-> STM Velocity/Velocity
//   (this object) <-> Device 1 (EtherCAT)/Term 5 (EK1200)/Term 6 (EK1122-0080)/DRL02-EK0 (EK1101-0080)/DRL02-E12 (EL5042)
//     Enc/Inputs/In/nComState @bit 1 <-> WcState/InputToggle
//     Enc/Inputs/In/nComState <-> WcState/WcState
//     Enc/Inputs/In/nDataIn1 <-> FB Inputs Channel 1/Position
//     Enc/Inputs/In/nDataIn1 <-> FB Inputs Channel 2/Position
//     Enc/Inputs/In/nState1 @bit 12 <-> FB Inputs Channel 1/Status/Diag
//     Enc/Inputs/In/nState1 @bit 12 <-> FB Inputs Channel 2/Status/Diag
//     Enc/Inputs/In/nState1 @bit 1 <-> FB Inputs Channel 1/Status/Error
//     Enc/Inputs/In/nState1 @bit 1 <-> FB Inputs Channel 2/Status/Error
//     Enc/Inputs/In/nState1 @bit 14 <-> FB Inputs Channel 1/Status/Input cycle counter
//     Enc/Inputs/In/nState1 @bit 14 <-> FB Inputs Channel 2/Status/Input cycle counter
//     Enc/Inputs/In/nState1 @bit 2 <-> FB Inputs Channel 1/Status/Ready
//     Enc/Inputs/In/nState1 @bit 2 <-> FB Inputs Channel 2/Status/Ready
//     Enc/Inputs/In/nState1 @bit 13 <-> FB Inputs Channel 1/Status/TxPDO State
//     Enc/Inputs/In/nState1 @bit 13 <-> FB Inputs Channel 2/Status/TxPDO State
//     Enc/Inputs/In/nState1 <-> FB Inputs Channel 1/Status/Warning
//     Enc/Inputs/In/nState1 <-> FB Inputs Channel 2/Status/Warning
//   (this object) <-> Device 1 (EtherCAT)/Term 5 (EK1200)/Term 6 (EK1122-0080)/DRL02-EK0 (EK1101-0080)/DRL02-E13 (EL7041)
//     Drive/Inputs/In/nState1 @bit 3 <-> STM Status/Status/Error
//     Drive/Inputs/In/nState1 @bit 5 <-> STM Status/Status/Moving negative
//     Drive/Inputs/In/nState1 @bit 4 <-> STM Status/Status/Moving positive
//     Drive/Inputs/In/nState1 @bit 1 <-> STM Status/Status/Ready
//     Drive/Inputs/In/nState1 <-> STM Status/Status/Ready to enable
//     Drive/Inputs/In/nState1 @bit 6 <-> STM Status/Status/Torque reduced
//     Drive/Inputs/In/nState1 @bit 2 <-> STM Status/Status/Warning
//     Drive/Inputs/In/nState2 @bit 3 <-> STM Status/Status/Digital input 1
//     Drive/Inputs/In/nState2 @bit 4 <-> STM Status/Status/Digital input 2
//     Drive/Inputs/In/nState2 @bit 5 <-> STM Status/Status/Sync error
//     Drive/Inputs/In/nState2 @bit 7 <-> STM Status/Status/TxPDO Toggle
//     Drive/Inputs/In/nState4 @bit 1 <-> WcState/InputToggle
//     Drive/Inputs/In/nState4 <-> WcState/WcState
//     Drive/Outputs/Out/nCtrl1 <-> STM Control/Control/Enable
//     Drive/Outputs/Out/nCtrl1 @bit 2 <-> STM Control/Control/Reduce torque
//     Drive/Outputs/Out/nCtrl1 @bit 1 <-> STM Control/Control/Reset
//     Drive/Outputs/Out/nDataOut2[0] <-> STM Velocity/Velocity
//   (this object) <-> Device 1 (EtherCAT)/Term 5 (EK1200)/Term 6 (EK1122-0080)/DRL02-EK0 (EK1101-0080)/DRL02-E24 (EL7031)
//     Drive/Inputs/In/nState1 @bit 3 <-> STM Status/Status/Error
//     Drive/Inputs/In/nState1 @bit 5 <-> STM Status/Status/Moving negative
//     Drive/Inputs/In/nState1 @bit 4 <-> STM Status/Status/Moving positive
//     Drive/Inputs/In/nState1 @bit 1 <-> STM Status/Status/Ready
//     Drive/Inputs/In/nState1 <-> STM Status/Status/Ready to enable
//     Drive/Inputs/In/nState1 @bit 6 <-> STM Status/Status/Torque reduced
//     Drive/Inputs/In/nState1 @bit 2 <-> STM Status/Status/Warning
//     Drive/Inputs/In/nState2 @bit 3 <-> STM Status/Status/Digital input 1
//     Drive/Inputs/In/nState2 @bit 4 <-> STM Status/Status/Digital input 2
//     Drive/Inputs/In/nState2 @bit 5 <-> STM Status/Status/Sync error
//     Drive/Inputs/In/nState2 @bit 7 <-> STM Status/Status/TxPDO Toggle
//     Drive/Inputs/In/nState4 @bit 1 <-> WcState/InputToggle
//     Drive/Inputs/In/nState4 <-> WcState/WcState
//     Drive/Outputs/Out/nCtrl1 <-> STM Control/Control/Enable
//     Drive/Outputs/Out/nCtrl1 @bit 2 <-> STM Control/Control/Reduce torque
//     Drive/Outputs/Out/nCtrl1 @bit 1 <-> STM Control/Control/Reset
//     Drive/Outputs/Out/nDataOut2[0] <-> STM Velocity/Velocity
//   (this object) <-> Device 1 (EtherCAT)/Term 5 (EK1200)/Term 6 (EK1122-0080)/DRL02-EK0 (EK1101-0080)/Term 91 (EL5112)
//     Enc/Inputs/In/nDataIn1 <-> ENC Status Channel 1/Counter value
//     Enc/Inputs/In/nDataIn2 <-> ENC Status Channel 1/Latch value
//     Enc/Inputs/In/nState1 @bit 4 <-> ENC Status Channel 1/Status/Counter overflow
//     Enc/Inputs/In/nState1 @bit 3 <-> ENC Status Channel 1/Status/Counter underflow
//     Enc/Inputs/In/nState1 @bit 1 <-> ENC Status Channel 1/Status/Latch extern valid
//     Enc/Inputs/In/nState1 @bit 6 <-> ENC Status Channel 1/Status/Open circuit
//     Enc/Inputs/In/nState1 @bit 2 <-> ENC Status Channel 1/Status/Set counter done
//     Enc/Inputs/In/nState2 <-> ENC Status Channel 1/Status/Status of input A
//     Enc/Inputs/In/nState2 @bit 1 <-> ENC Status Channel 1/Status/Status of input B
//     Enc/Inputs/In/nState2 @bit 3 <-> ENC Status Channel 1/Status/Status of input gate
//     Enc/Inputs/In/nState4 @bit 1 <-> WcState/InputToggle
//     Enc/Inputs/In/nState4 <-> WcState/WcState
//     Enc/Outputs/Out/nCtrl1 @bit 3 <-> ENC Control Channel 1/Control/Enable latch extern on negative edge
//     Enc/Outputs/Out/nCtrl1 @bit 1 <-> ENC Control Channel 1/Control/Enable latch extern on positive edge
//     Enc/Outputs/Out/nCtrl1 @bit 2 <-> ENC Control Channel 1/Control/Set counter
//     Enc/Outputs/Out/nCtrl2 @bit 2 <-> ENC Control Channel 1/Control/Set counter on latch extern on negative edge
//     Enc/Outputs/Out/nCtrl2 @bit 1 <-> ENC Control Channel 1/Control/Set counter on latch extern on positive edge
//     Enc/Outputs/Out/nCtrl2 <-> ENC Control Channel 1/Control/Set software gate
//     Enc/Outputs/Out/nDataOut1 <-> ENC Control Channel 1/Set counter value
//   (this object) <-> Device 1 (EtherCAT)/Term 5 (EK1200)/Term 6 (EK1122-0080)/DRL02-EK0 (EK1101-0080)/DRL02-E25 (EL5042)
//     Enc/Inputs/In/nComState @bit 1 <-> WcState/InputToggle
//     Enc/Inputs/In/nComState <-> WcState/WcState
//     Enc/Inputs/In/nDataIn1 <-> FB Inputs Channel 2/Position
//     Enc/Inputs/In/nState1 @bit 12 <-> FB Inputs Channel 2/Status/Diag
//     Enc/Inputs/In/nState1 @bit 1 <-> FB Inputs Channel 2/Status/Error
//     Enc/Inputs/In/nState1 @bit 14 <-> FB Inputs Channel 2/Status/Input cycle counter
//     Enc/Inputs/In/nState1 @bit 2 <-> FB Inputs Channel 2/Status/Ready
//     Enc/Inputs/In/nState1 @bit 13 <-> FB Inputs Channel 2/Status/TxPDO State
//     Enc/Inputs/In/nState1 <-> FB Inputs Channel 2/Status/Warning
//   (this object) <-> Device 1 (EtherCAT)/Term 5 (EK1200)/Term 6 (EK1122-0080)/DRL02-EK0 (EK1101-0080)/DRL02-E26 (EL7031)
//     Drive/Inputs/In/nState1 @bit 3 <-> STM Status/Status/Error
//     Drive/Inputs/In/nState1 @bit 5 <-> STM Status/Status/Moving negative
//     Drive/Inputs/In/nState1 @bit 4 <-> STM Status/Status/Moving positive
//     Drive/Inputs/In/nState1 @bit 1 <-> STM Status/Status/Ready
//     Drive/Inputs/In/nState1 <-> STM Status/Status/Ready to enable
//     Drive/Inputs/In/nState1 @bit 6 <-> STM Status/Status/Torque reduced
//     Drive/Inputs/In/nState1 @bit 2 <-> STM Status/Status/Warning
//     Drive/Inputs/In/nState2 @bit 3 <-> STM Status/Status/Digital input 1
//     Drive/Inputs/In/nState2 @bit 4 <-> STM Status/Status/Digital input 2
//     Drive/Inputs/In/nState2 @bit 5 <-> STM Status/Status/Sync error
//     Drive/Inputs/In/nState2 @bit 7 <-> STM Status/Status/TxPDO Toggle
//     Drive/Inputs/In/nState4 @bit 1 <-> WcState/InputToggle
//     Drive/Inputs/In/nState4 <-> WcState/WcState
//     Drive/Outputs/Out/nCtrl1 <-> STM Control/Control/Enable
//     Drive/Outputs/Out/nCtrl1 @bit 2 <-> STM Control/Control/Reduce torque
//     Drive/Outputs/Out/nCtrl1 @bit 1 <-> STM Control/Control/Reset
//     Drive/Outputs/Out/nDataOut2[0] <-> STM Velocity/Velocity
//   (this object) <-> Device 1 (EtherCAT)/Term 5 (EK1200)/Term 6 (EK1122-0080)/DRL02-EK0 (EK1101-0080)/DRL02-E28 (EL5042)
//     Enc/Inputs/In/nComState @bit 1 <-> WcState/InputToggle
//     Enc/Inputs/In/nComState <-> WcState/WcState
//     Enc/Inputs/In/nDataIn1 <-> FB Inputs Channel 2/Position
//     Enc/Inputs/In/nDataIn1 <-> FB Inputs Channel 1/Position
//     Enc/Inputs/In/nState1 @bit 12 <-> FB Inputs Channel 2/Diag
//     Enc/Inputs/In/nState1 @bit 1 <-> FB Inputs Channel 2/Error
//     Enc/Inputs/In/nState1 @bit 14 <-> FB Inputs Channel 2/Input cycle counter
//     Enc/Inputs/In/nState1 @bit 2 <-> FB Inputs Channel 2/Ready
//     Enc/Inputs/In/nState1 @bit 13 <-> FB Inputs Channel 2/TxPDO State
//     Enc/Inputs/In/nState1 <-> FB Inputs Channel 2/Warning
//   (this object) <-> Device 1 (EtherCAT)/Term 5 (EK1200)/Term 6 (EK1122-0080)/DRL02-EK0 (EK1101-0080)/DRL02-E29 (EL7031)
//     Drive/Inputs/In/nState1 @bit 3 <-> STM Status/Status/Error
//     Drive/Inputs/In/nState1 @bit 5 <-> STM Status/Status/Moving negative
//     Drive/Inputs/In/nState1 @bit 4 <-> STM Status/Status/Moving positive
//     Drive/Inputs/In/nState1 @bit 1 <-> STM Status/Status/Ready
//     Drive/Inputs/In/nState1 <-> STM Status/Status/Ready to enable
//     Drive/Inputs/In/nState1 @bit 6 <-> STM Status/Status/Torque reduced
//     Drive/Inputs/In/nState1 @bit 2 <-> STM Status/Status/Warning
//     Drive/Inputs/In/nState2 @bit 3 <-> STM Status/Status/Digital input 1
//     Drive/Inputs/In/nState2 @bit 4 <-> STM Status/Status/Digital input 2
//     Drive/Inputs/In/nState2 @bit 5 <-> STM Status/Status/Sync error
//     Drive/Inputs/In/nState2 @bit 7 <-> STM Status/Status/TxPDO Toggle
//     Drive/Inputs/In/nState4 @bit 1 <-> WcState/InputToggle
//     Drive/Inputs/In/nState4 <-> WcState/WcState
//     Drive/Outputs/Out/nCtrl1 <-> STM Control/Control/Enable
//     Drive/Outputs/Out/nCtrl1 @bit 2 <-> STM Control/Control/Reduce torque
//     Drive/Outputs/Out/nCtrl1 @bit 1 <-> STM Control/Control/Reset
//     Drive/Outputs/Out/nDataOut2[0] <-> STM Velocity/Velocity
//   (this object) <-> Device 1 (EtherCAT)/Term 5 (EK1200)/Term 6 (EK1122-0080)/DRL02-EK0 (EK1101-0080)/DRL02-E30 (EL7031)
//     Drive/Inputs/In/nState1 @bit 3 <-> STM Status/Status/Error
//     Drive/Inputs/In/nState1 @bit 5 <-> STM Status/Status/Moving negative
//     Drive/Inputs/In/nState1 @bit 4 <-> STM Status/Status/Moving positive
//     Drive/Inputs/In/nState1 @bit 1 <-> STM Status/Status/Ready
//     Drive/Inputs/In/nState1 <-> STM Status/Status/Ready to enable
//     Drive/Inputs/In/nState1 @bit 6 <-> STM Status/Status/Torque reduced
//     Drive/Inputs/In/nState1 @bit 2 <-> STM Status/Status/Warning
//     Drive/Inputs/In/nState2 @bit 3 <-> STM Status/Status/Digital input 1
//     Drive/Inputs/In/nState2 @bit 4 <-> STM Status/Status/Digital input 2
//     Drive/Inputs/In/nState2 @bit 5 <-> STM Status/Status/Sync error
//     Drive/Inputs/In/nState2 @bit 7 <-> STM Status/Status/TxPDO Toggle
//     Drive/Inputs/In/nState4 @bit 1 <-> WcState/InputToggle
//     Drive/Inputs/In/nState4 <-> WcState/WcState
//     Drive/Outputs/Out/nCtrl1 <-> STM Control/Control/Enable
//     Drive/Outputs/Out/nCtrl1 @bit 2 <-> STM Control/Control/Reduce torque
//     Drive/Outputs/Out/nCtrl1 @bit 1 <-> STM Control/Control/Reset
//     Drive/Outputs/Out/nDataOut2[0] <-> STM Velocity/Velocity
//     Enc/Inputs/In/nDataIn1[0] <-> ENC Status compact/Counter value
//     Enc/Inputs/In/nDataIn2[0] <-> ENC Status compact/Latch value
//     Enc/Inputs/In/nState1 @bit 4 <-> ENC Status compact/Status/Counter overflow
//     Enc/Inputs/In/nState1 @bit 3 <-> ENC Status compact/Status/Counter underflow
//     Enc/Inputs/In/nState1 @bit 1 <-> ENC Status compact/Status/Latch extern valid
//     Enc/Inputs/In/nState1 @bit 2 <-> ENC Status compact/Status/Set counter done
//     Enc/Inputs/In/nState2 @bit 4 <-> ENC Status compact/Status/Status of extern latch
//     Enc/Inputs/In/nState2 @bit 5 <-> ENC Status compact/Status/Sync error
//     Enc/Inputs/In/nState2 @bit 7 <-> ENC Status compact/Status/TxPDO Toggle
//     Enc/Inputs/In/nState4 @bit 1 <-> WcState/InputToggle
//     Enc/Inputs/In/nState4 <-> WcState/WcState
//     Enc/Outputs/Out/nCtrl1 @bit 3 <-> ENC Control compact/Control/Enable latch extern on negative edge
//     Enc/Outputs/Out/nCtrl1 @bit 1 <-> ENC Control compact/Control/Enable latch extern on positive edge
//     Enc/Outputs/Out/nCtrl1 @bit 2 <-> ENC Control compact/Control/Set counter
//     Enc/Outputs/Out/nDataOut1[0] <-> ENC Control compact/Set counter value
//   (this object) <-> Device 1 (EtherCAT)/Term 5 (EK1200)/Term 6 (EK1122-0080)/DRL02-EK0 (EK1101-0080)/DRL02-E31 (EL7031)
//     Drive/Inputs/In/nState1 @bit 3 <-> STM Status/Status/Error
//     Drive/Inputs/In/nState1 @bit 5 <-> STM Status/Status/Moving negative
//     Drive/Inputs/In/nState1 @bit 4 <-> STM Status/Status/Moving positive
//     Drive/Inputs/In/nState1 @bit 1 <-> STM Status/Status/Ready
//     Drive/Inputs/In/nState1 <-> STM Status/Status/Ready to enable
//     Drive/Inputs/In/nState1 @bit 6 <-> STM Status/Status/Torque reduced
//     Drive/Inputs/In/nState1 @bit 2 <-> STM Status/Status/Warning
//     Drive/Inputs/In/nState2 @bit 3 <-> STM Status/Status/Digital input 1
//     Drive/Inputs/In/nState2 @bit 4 <-> STM Status/Status/Digital input 2
//     Drive/Inputs/In/nState2 @bit 5 <-> STM Status/Status/Sync error
//     Drive/Inputs/In/nState2 @bit 7 <-> STM Status/Status/TxPDO Toggle
//     Drive/Inputs/In/nState4 @bit 1 <-> WcState/InputToggle
//     Drive/Inputs/In/nState4 <-> WcState/WcState
//     Drive/Outputs/Out/nCtrl1 <-> STM Control/Control/Enable
//     Drive/Outputs/Out/nCtrl1 @bit 2 <-> STM Control/Control/Reduce torque
//     Drive/Outputs/Out/nCtrl1 @bit 1 <-> STM Control/Control/Reset
//     Drive/Outputs/Out/nDataOut2[0] <-> STM Velocity/Velocity
//   (this object) <-> Device 1 (EtherCAT)/Term 5 (EK1200)/Term 6 (EK1122-0080)/DRL02-EK0 (EK1101-0080)/DRL02-E32 (EL5042)
//     Enc/Inputs/In/nComState @bit 1 <-> WcState/InputToggle
//     Enc/Inputs/In/nComState <-> WcState/WcState
//     Enc/Inputs/In/nDataIn1 <-> FB Inputs Channel 1/Position
//     Enc/Inputs/In/nState1 @bit 12 <-> FB Inputs Channel 1/Status/Diag
//     Enc/Inputs/In/nState1 @bit 1 <-> FB Inputs Channel 1/Status/Error
//     Enc/Inputs/In/nState1 @bit 14 <-> FB Inputs Channel 1/Status/Input cycle counter
//     Enc/Inputs/In/nState1 @bit 2 <-> FB Inputs Channel 1/Status/Ready
//     Enc/Inputs/In/nState1 @bit 13 <-> FB Inputs Channel 1/Status/TxPDO State
//     Enc/Inputs/In/nState1 <-> FB Inputs Channel 1/Status/Warning
//   PLC_CRIX_MOT Instance <-> Device 1 (EtherCAT)/Term 5 (EK1200)/Term 167 (EK1122)/CRIX_VAC_INTF (EL6695-0002)
//     PlcTask Inputs/PRG_CryoPump.bCRYO_VGC_01_CLS <-> IO Inputs/bCRYO_VGC_01_CLS
//     PlcTask Inputs/PRG_CryoPump.bCRYO_VGC_02_CLS <-> IO Inputs/bCRYO_VGC_02_CLS
//     PlcTask Inputs/PRG_CryoPump.bCRYO_VGC_01_OPN <-> IO Inputs/bCRYO_VGC_01_OPN
//     PlcTask Inputs/PRG_CryoPump.bCRYO_VGC_02_OPN <-> IO Inputs/bCRYO_VGC_02_OPN
//     PlcTask Inputs/PRG_CryoPump.xEcatBridge_External_device_not_connected <-> SYNC Inputs/External device not connected
//     PlcTask Inputs/PRG_CryoPump.xEcatBridge_TxPDO_state <-> SYNC Inputs/TxPDO state
//     PlcTask Inputs/PRG_CryoPump.xEcatBridge_WcState <-> WcState/WcState
//     PlcTask Inputs/PRG_InjectorMotors.bSDS_VGC_01_CLS <-> IO Inputs/bSDS_VGC_01_CLS
//     PlcTask Inputs/PRG_InjectorMotors.bSDS_VGC_01_OPN <-> IO Inputs/bSDS_VGC_01_OPN
//     PlcTask Outputs/PRG_CryoPump.bMOTY10_IN <-> IO Outputs/bMOTY10_IN
//     PlcTask Outputs/PRG_CryoPump.bMOTY11_IN <-> IO Outputs/bMOTY11_IN
//     PlcTask Outputs/PRG_CryoPump.bMOTY10_OUT <-> IO Outputs/bMOTY10_OUT
//     PlcTask Outputs/PRG_CryoPump.bMOTY11_OUT <-> IO Outputs/bMOTY11_OUT
//     PlcTask Outputs/PRG_InjectorMotors.bMOTSDSZ18_IN <-> IO Outputs/bMOTSDSZ18_IN
//     PlcTask Outputs/PRG_InjectorMotors.bMOTSDSZ18_OUT <-> IO Outputs/bMOTSDSZ18_OUT
//   PLC_CRIX_MOT Instance <-> Device 1 (EtherCAT)/Term 5 (EK1200)/Term 6 (EK1122-0080)/DRL02-EK0 (EK1101-0080)/DRL02-E1 (EL7031)
//     PlcTask Inputs/Main.M1.bLimitBackwardEnable <-> STM Status/Status/Digital input 1
//     PlcTask Inputs/Main.M1.bLimitForwardEnable <-> STM Status/Status/Digital input 2
//   PLC_CRIX_MOT Instance <-> Device 1 (EtherCAT)/Term 5 (EK1200)/Term 6 (EK1122-0080)/DRL02-EK0 (EK1101-0080)/DRL02-E11 (EL7031)
//     PlcTask Inputs/Main.M7.bLimitBackwardEnable <-> STM Status/Status/Digital input 2
//     PlcTask Inputs/Main.M7.bLimitForwardEnable <-> STM Status/Status/Digital input 1
//   PLC_CRIX_MOT Instance <-> Device 1 (EtherCAT)/Term 5 (EK1200)/Term 6 (EK1122-0080)/DRL02-EK0 (EK1101-0080)/DRL02-E13 (EL7041)
//     PlcTask Inputs/Main.M8.bLimitBackwardEnable <-> STM Status/Status/Digital input 2
//     PlcTask Inputs/Main.M8.bLimitForwardEnable <-> STM Status/Status/Digital input 1
//   PLC_CRIX_MOT Instance <-> Device 1 (EtherCAT)/Term 5 (EK1200)/Term 6 (EK1122-0080)/DRL02-EK0 (EK1101-0080)/DRL02-E17 (EL7031)
//     PlcTask Inputs/Main.M12.bLimitBackwardEnable <-> STM Status/Status/Digital input 2
//     PlcTask Inputs/Main.M12.bLimitForwardEnable <-> STM Status/Status/Digital input 1
//   PLC_CRIX_MOT Instance <-> Device 1 (EtherCAT)/Term 5 (EK1200)/Term 6 (EK1122-0080)/DRL02-EK0 (EK1101-0080)/DRL02-E19 (EL7031)
//     PlcTask Inputs/Main.M13.bLimitBackwardEnable <-> STM Status/Status/Digital input 2
//     PlcTask Inputs/Main.M13.bLimitForwardEnable <-> STM Status/Status/Digital input 1
//   PLC_CRIX_MOT Instance <-> Device 1 (EtherCAT)/Term 5 (EK1200)/Term 6 (EK1122-0080)/DRL02-EK0 (EK1101-0080)/DRL02-E21 (EL7041)
//     PlcTask Inputs/Main.M49.bLimitForwardEnable <-> STM Status/Status/Digital input 2
//     PlcTask Inputs/PRG_CryoPump.bLimitBackwardEnable_Y_11 <-> STM Status/Status/Digital input 1
//   PLC_CRIX_MOT Instance <-> Device 1 (EtherCAT)/Term 5 (EK1200)/Term 6 (EK1122-0080)/DRL02-EK0 (EK1101-0080)/DRL02-E23 (EL7041)
//     PlcTask Inputs/Main.M48.bLimitForwardEnable <-> STM Status/Status/Digital input 2
//     PlcTask Inputs/PRG_CryoPump.bLimitBackwardEnable_Y_10 <-> STM Status/Status/Digital input 1
//   PLC_CRIX_MOT Instance <-> Device 1 (EtherCAT)/Term 5 (EK1200)/Term 6 (EK1122-0080)/DRL02-EK0 (EK1101-0080)/DRL02-E26 (EL7031)
//     PlcTask Inputs/Main.M17.bLimitBackwardEnable <-> STM Status/Status/Digital input 2
//     PlcTask Inputs/Main.M17.bLimitForwardEnable <-> STM Status/Status/Digital input 1
//   PLC_CRIX_MOT Instance <-> Device 1 (EtherCAT)/Term 5 (EK1200)/Term 6 (EK1122-0080)/DRL02-EK0 (EK1101-0080)/DRL02-E27 (EL7031)
//     PlcTask Inputs/Main.M18.bLimitForwardEnable <-> STM Status/Status/Digital input 1
//     PlcTask Inputs/PRG_InjectorMotors.bLimitBackwardEnable_SDSZ_18 <-> STM Status/Status/Digital input 2
//   PLC_CRIX_MOT Instance <-> Device 1 (EtherCAT)/Term 5 (EK1200)/Term 6 (EK1122-0080)/DRL02-EK0 (EK1101-0080)/DRL02-E3 (EL7031)
//     PlcTask Inputs/Main.M2.bLimitBackwardEnable <-> STM Status/Status/Digital input 2
//     PlcTask Inputs/Main.M2.bLimitForwardEnable <-> STM Status/Status/Digital input 1
//   PLC_CRIX_MOT Instance <-> Device 1 (EtherCAT)/Term 5 (EK1200)/Term 6 (EK1122-0080)/DRL02-EK0 (EK1101-0080)/DRL02-E31 (EL7031)
//     PlcTask Inputs/Main.M35.bLimitBackwardEnable <-> STM Status/Status/Digital input 2
//     PlcTask Inputs/Main.M35.bLimitForwardEnable <-> STM Status/Status/Digital input 1
//   PLC_CRIX_MOT Instance <-> Device 1 (EtherCAT)/Term 5 (EK1200)/Term 6 (EK1122-0080)/DRL02-EK0 (EK1101-0080)/DRL02-E4 (EL7031)
//     PlcTask Inputs/Main.M3.bLimitBackwardEnable <-> STM Status/Status/Digital input 2
//     PlcTask Inputs/Main.M3.bLimitForwardEnable <-> STM Status/Status/Digital input 1
//   PLC_CRIX_MOT Instance <-> Device 1 (EtherCAT)/Term 5 (EK1200)/Term 6 (EK1122-0080)/DRL02-EK0 (EK1101-0080)/DRL02-E6 (EL7031)
//     PlcTask Inputs/Main.M4.bLimitBackwardEnable <-> STM Status/Status/Digital input 1
//     PlcTask Inputs/Main.M4.bLimitForwardEnable <-> STM Status/Status/Digital input 2
//   PLC_CRIX_MOT Instance <-> Device 1 (EtherCAT)/Term 5 (EK1200)/Term 6 (EK1122-0080)/DRL02-EK0 (EK1101-0080)/DRL02-E7 (EL7031)
//     PlcTask Inputs/Main.M5.bLimitBackwardEnable <-> STM Status/Status/Digital input 2
//     PlcTask Inputs/Main.M5.bLimitForwardEnable <-> STM Status/Status/Digital input 1
//   PLC_CRIX_MOT Instance <-> Device 1 (EtherCAT)/Term 5 (EK1200)/Term 6 (EK1122-0080)/DRL02-EK0 (EK1101-0080)/DRL02-E9 (EL7031)
//     PlcTask Inputs/Main.M6.bLimitBackwardEnable <-> STM Status/Status/Digital input 2
//     PlcTask Inputs/Main.M6.bLimitForwardEnable <-> STM Status/Status/Digital input 1
//   PLC_CRIX_MOT Instance <-> Device 1 (EtherCAT)/Term 5 (EK1200)/Term 6 (EK1122-0080)/DRL02-EK0 (EK1101-0080)/DRL02-ECJ0 (EK1122-0080)/Term 109 (EK1101-0080)/Camera X (EL7041)
//     PlcTask Inputs/Main.M33.bLimitBackwardEnable <-> STM Status/Status/Digital input 2
//     PlcTask Inputs/Main.M33.bLimitForwardEnable <-> STM Status/Status/Digital input 1
//   PLC_CRIX_MOT Instance <-> Device 1 (EtherCAT)/Term 5 (EK1200)/Term 6 (EK1122-0080)/DRL02-EK0 (EK1101-0080)/DRL02-ECJ0 (EK1122-0080)/Term 109 (EK1101-0080)/Camera Y (EL7041)
//     PlcTask Inputs/Main.M34.bLimitBackwardEnable <-> STM Status/Status/Digital input 2
//     PlcTask Inputs/Main.M34.bLimitForwardEnable <-> STM Status/Status/Digital input 1
//   PLC_CRIX_MOT Instance <-> Device 1 (EtherCAT)/Term 5 (EK1200)/Term 6 (EK1122-0080)/DRL02-EK0 (EK1101-0080)/DRL02-ECJ0 (EK1122-0080)/Term 113 (EK1101-0080)/FZP X (EL7041)
//     PlcTask Inputs/Main.M31.bLimitBackwardEnable <-> STM Status/Status/Digital input 2
//     PlcTask Inputs/Main.M31.bLimitForwardEnable <-> STM Status/Status/Digital input 1
//   PLC_CRIX_MOT Instance <-> Device 1 (EtherCAT)/Term 5 (EK1200)/Term 6 (EK1122-0080)/DRL02-EK0 (EK1101-0080)/DRL02-ECJ0 (EK1122-0080)/Term 113 (EK1101-0080)/FZP Y (EL7041)
//     PlcTask Inputs/Main.M30.bLimitBackwardEnable <-> STM Status/Status/Digital input 2
//     PlcTask Inputs/Main.M30.bLimitForwardEnable <-> STM Status/Status/Digital input 1
//   PLC_CRIX_MOT Instance <-> Device 1 (EtherCAT)/Term 5 (EK1200)/Term 6 (EK1122-0080)/DRL02-EK0 (EK1101-0080)/DRL02-ECJ0 (EK1122-0080)/Term 113 (EK1101-0080)/FZP Z (EL7041)
//     PlcTask Inputs/Main.M32.bLimitBackwardEnable <-> STM Status/Status/Digital input 2
//     PlcTask Inputs/Main.M32.bLimitForwardEnable <-> STM Status/Status/Digital input 1
//   PLC_CRIX_MOT Instance <-> Device 1 (EtherCAT)/Term 5 (EK1200)/Term 6 (EK1122-0080)/DRL02-EK0 (EK1101-0080)/DRL02-ECJ1 (EK1122)/CryoStat (EK1101)/Cryo X (EL7041)
//     PlcTask Inputs/Main.M22.bLimitBackwardEnable <-> STM Status/Status/Digital input 2
//     PlcTask Inputs/Main.M22.bLimitForwardEnable <-> STM Status/Status/Digital input 1
//   PLC_CRIX_MOT Instance <-> Device 1 (EtherCAT)/Term 5 (EK1200)/Term 6 (EK1122-0080)/DRL02-EK0 (EK1101-0080)/DRL02-ECJ1 (EK1122)/CryoStat (EK1101)/Cryo Y (EL7041)
//     PlcTask Inputs/Main.M23.bLimitBackwardEnable <-> STM Status/Status/Digital input 2
//     PlcTask Inputs/Main.M23.bLimitForwardEnable <-> STM Status/Status/Digital input 1
//   PLC_CRIX_MOT Instance <-> Device 1 (EtherCAT)/Term 5 (EK1200)/Term 6 (EK1122-0080)/DRL02-EK0 (EK1101-0080)/DRL02-ECJ1 (EK1122)/CryoStat (EK1101)/Cryo Z (EL7041)
//     PlcTask Inputs/Main.M24.bLimitBackwardEnable <-> STM Status/Status/Digital input 2
//     PlcTask Inputs/Main.M24.bLimitForwardEnable <-> STM Status/Status/Digital input 1
//   PLC_CRIX_MOT Instance <-> Device 1 (EtherCAT)/Term 5 (EK1200)/Term 6 (EK1122-0080)/DRL02-EK0 (EK1101-0080)/DRL02-ECJ1 (EK1122)/CryoStat (EK1101)/FiberLite (EL4004)
//     PlcTask Outputs/GVL_FiberLite.bLedOutput2.iIlluminatorINT <-> AO Outputs Channel 2/Analog output
//     PlcTask Outputs/GVL_FiberLite.bLedOutput3.iIlluminatorINT <-> AO Outputs Channel 3/Analog output
//     PlcTask Outputs/GVL_FiberLite.bLedOutput4.iIlluminatorINT <-> AO Outputs Channel 4/Analog output
//   PLC_CRIX_MOT Instance <-> Device 1 (EtherCAT)/Term 5 (EK1200)/Term 6 (EK1122-0080)/DRL02-EK0 (EK1101-0080)/DRL02-ECJ1 (EK1122)/VLS_EP10_EP7041-3102
//     PlcTask Inputs/Main.M44.bHome <-> ENC Status compact/Status/Status of input C
//     PlcTask Inputs/Main.M44.bLimitBackwardEnable <-> STM Status/Status/Digital input 1
//     PlcTask Inputs/Main.M44.bLimitForwardEnable <-> STM Status/Status/Digital input 2
//     PlcTask Inputs/Main.M44.nRawEncoderUINT <-> ENC Status compact/Counter value
//   PLC_CRIX_MOT Instance <-> Device 1 (EtherCAT)/Term 5 (EK1200)/Term 6 (EK1122-0080)/DRL02-EK0 (EK1101-0080)/DRL02-ECJ1 (EK1122)/VLS_EP11_EP7041-3102
//     PlcTask Inputs/Main.M45.bHome <-> ENC Status compact/Status/Status of input C
//     PlcTask Inputs/Main.M45.bLimitBackwardEnable <-> STM Status/Status/Digital input 1
//     PlcTask Inputs/Main.M45.bLimitForwardEnable <-> STM Status/Status/Digital input 2
//     PlcTask Inputs/Main.M45.nRawEncoderUINT <-> ENC Status compact/Counter value
//   PLC_CRIX_MOT Instance <-> Device 1 (EtherCAT)/Term 5 (EK1200)/Term 6 (EK1122-0080)/DRL02-EK0 (EK1101-0080)/DRL02-ECJ1 (EK1122)/VLS_EP12_EP7041-3102
//     PlcTask Inputs/Main.M46.bHome <-> ENC Status compact/Status/Status of input C
//     PlcTask Inputs/Main.M46.bLimitBackwardEnable <-> STM Status/Status/Digital input 2
//     PlcTask Inputs/Main.M46.bLimitForwardEnable <-> STM Status/Status/Digital input 1
//   PLC_CRIX_MOT Instance <-> Device 1 (EtherCAT)/Term 5 (EK1200)/Term 6 (EK1122-0080)/DRL02-EK0 (EK1101-0080)/DRL02-ECJ1 (EK1122)/VLS_EP13_EP7041-3102
//     PlcTask Inputs/Main.M47.bHome <-> ENC Status compact/Status/Status of input C
//     PlcTask Inputs/Main.M47.bLimitBackwardEnable <-> STM Status/Status/Digital input 1
//     PlcTask Inputs/Main.M47.bLimitForwardEnable <-> STM Status/Status/Digital input 2
//   PLC_CRIX_MOT Instance <-> Device 1 (EtherCAT)/Term 5 (EK1200)/Term 6 (EK1122-0080)/DRL02-EK0 (EK1101-0080)/DRL02-ECJ1 (EK1122)/VLS_EP6_EP7041-1002
//     PlcTask Inputs/Main.M40.bLimitBackwardEnable <-> STM Status/Status/Digital input 2
//     PlcTask Inputs/Main.M40.bLimitForwardEnable <-> STM Status/Status/Digital input 1
//   PLC_CRIX_MOT Instance <-> Device 1 (EtherCAT)/Term 5 (EK1200)/Term 6 (EK1122-0080)/DRL02-EK0 (EK1101-0080)/DRL02-ECJ1 (EK1122)/VLS_EP7_EP7041-1002
//     PlcTask Inputs/Main.M41.bLimitBackwardEnable <-> STM Status/Status/Digital input 2
//     PlcTask Inputs/Main.M41.bLimitForwardEnable <-> STM Status/Status/Digital input 1
//   PLC_CRIX_MOT Instance <-> Device 1 (EtherCAT)/Term 5 (EK1200)/Term 6 (EK1122-0080)/DRL02-EK0 (EK1101-0080)/DRL02-ECJ1 (EK1122)/VLS_EP8_EP7041-1002
//     PlcTask Inputs/Main.M42.bLimitBackwardEnable <-> STM Status/Status/Digital input 2
//     PlcTask Inputs/Main.M42.bLimitForwardEnable <-> STM Status/Status/Digital input 1
//   PLC_CRIX_MOT Instance <-> Device 1 (EtherCAT)/Term 5 (EK1200)/Term 6 (EK1122-0080)/DRL02-EK0 (EK1101-0080)/DRL02-ECJ1 (EK1122)/VLS_EP9_EP7041-1002
//     PlcTask Inputs/Main.M43.bLimitBackwardEnable <-> STM Status/Status/Digital input 2
//     PlcTask Inputs/Main.M43.bLimitForwardEnable <-> STM Status/Status/Digital input 1
//   PLC_CRIX_MOT Instance <-> Device 1 (EtherCAT)/Term 5 (EK1200)/Term 6 (EK1122-0080)/DRL02-EK0 (EK1101-0080)/DRL02-ECJ2 (EK1122)/Catcher (EK1100)/Catcher_E1_EL7041
//     PlcTask Inputs/Main.M37.bLimitBackwardEnable <-> STM Status/Status/Digital input 1
//     PlcTask Inputs/Main.M37.bLimitForwardEnable <-> STM Status/Status/Digital input 2
//   PLC_CRIX_MOT Instance <-> Device 1 (EtherCAT)/Term 5 (EK1200)/Term 6 (EK1122-0080)/DRL02-EK0 (EK1101-0080)/DRL02-ECJ2 (EK1122)/Catcher (EK1100)/Catcher_E3_EL7041
//     PlcTask Inputs/Main.M38.bLimitBackwardEnable <-> STM Status/Status/Digital input 2
//     PlcTask Inputs/Main.M38.bLimitForwardEnable <-> STM Status/Status/Digital input 1
//   PLC_CRIX_MOT Instance <-> Device 1 (EtherCAT)/Term 5 (EK1200)/Term 6 (EK1122-0080)/DRL02-EK0 (EK1101-0080)/DRL02-ECJ2 (EK1122)/Catcher (EK1100)/Catcher_E4_EL7041
//     PlcTask Inputs/Main.M39.bLimitBackwardEnable <-> STM Status/Status/Digital input 1
//     PlcTask Inputs/Main.M39.bLimitForwardEnable <-> STM Status/Status/Digital input 2
//   PLC_CRIX_MOT Instance <-> Device 1 (EtherCAT)/Term 5 (EK1200)/Term 6 (EK1122-0080)/DRL02-EK0 (EK1101-0080)/Term 173 (EL1124)
//     PlcTask Inputs/PRG_InjectorMotors.bHall_Backward <-> Channel 4/Input
//     PlcTask Inputs/PRG_InjectorMotors.bHall_Forward <-> Channel 3/Input
//   PLC_CRIX_MOT Instance <-> Device 1 (EtherCAT)/Term 5 (EK1200)/Term 6 (EK1122-0080)/DRL02-EK0 (EK1101-0080)/Term 65 (EL1084)
//     PlcTask Inputs/Main.M10.bLimitBackwardEnable <-> Channel 4/Input
//     PlcTask Inputs/Main.M9.bLimitBackwardEnable <-> Channel 2/Input
//     PlcTask Inputs/Main.M10.bLimitForwardEnable <-> Channel 3/Input
//     PlcTask Inputs/Main.M9.bLimitForwardEnable <-> Channel 1/Input
//   PLC_CRIX_MOT Instance <-> Device 1 (EtherCAT)/Term 5 (EK1200)/Term 6 (EK1122-0080)/DRL02-EK0 (EK1101-0080)/Term 68 (EL1084)
//     PlcTask Inputs/Main.M11.bLimitBackwardEnable <-> Channel 2/Input
//     PlcTask Inputs/Main.M11.bLimitForwardEnable <-> Channel 1/Input
//   PLC_CRIX_MOT Instance <-> Device 1 (EtherCAT)/Term 5 (EK1200)/Term 83 (EK1521-0010)/Term 166 (EK1501-0010)/PMPS_FFO
//     PlcTask Outputs/GVL_PMPS.g_FastFaultOutput1.q_xFastFaultOut <-> Channel 1/Output
//     PlcTask Outputs/GVL_PMPS.g_FastFaultOutput2.q_xFastFaultOut <-> Channel 2/Output
//   PLC_CRIX_MOT Instance <-> Device 1 (EtherCAT)/Term 5 (EK1200)/Term 83 (EK1521-0010)/Term 166 (EK1501-0010)/PMPS_PRE
//     PlcTask Inputs/PRG_PMPS.fbArbiterIO.i_stCurrentBP <-> IO Inputs/CurrentBP
//     PlcTask Inputs/PRG_PMPS.fbArbiterIO.xTxPDO_state <-> SYNC Inputs/TxPDO state
//     PlcTask Inputs/PRG_PMPS.fbArbiterIO.xTxPDO_toggle <-> SYNC Inputs/TxPDO toggle
//     PlcTask Outputs/PRG_PMPS.fbArbiterIO.q_stRequestedBP <-> IO Outputs/RequestedBP
//   PLC_CRIX_MOT Instance <-> NC-Task 1 SAF/Axes/Axis 1 - Diagnostic Paddle X
//     PlcTask Inputs/Main.M1.Axis.NcToPlc <-> Outputs/ToPlc
//     PlcTask Outputs/Main.M1.Axis.PlcToNc <-> Inputs/FromPlc
//   PLC_CRIX_MOT Instance <-> NC-Task 1 SAF/Axes/Axis 10 - Illumination Y
//     PlcTask Inputs/Main.M10.Axis.NcToPlc <-> Outputs/ToPlc
//     PlcTask Outputs/Main.M10.Axis.PlcToNc <-> Inputs/FromPlc
//   PLC_CRIX_MOT Instance <-> NC-Task 1 SAF/Axes/Axis 11 - Illumination Z
//     PlcTask Inputs/Main.M11.Axis.NcToPlc <-> Outputs/ToPlc
//     PlcTask Outputs/Main.M11.Axis.PlcToNc <-> Inputs/FromPlc
//   PLC_CRIX_MOT Instance <-> NC-Task 1 SAF/Axes/Axis 12 - Questar X
//     PlcTask Inputs/Main.M12.Axis.NcToPlc <-> Outputs/ToPlc
//     PlcTask Outputs/Main.M12.Axis.PlcToNc <-> Inputs/FromPlc
//   PLC_CRIX_MOT Instance <-> NC-Task 1 SAF/Axes/Axis 13 - Questar Y
//     PlcTask Inputs/Main.M13.Axis.NcToPlc <-> Outputs/ToPlc
//     PlcTask Outputs/Main.M13.Axis.PlcToNc <-> Inputs/FromPlc
//   PLC_CRIX_MOT Instance <-> NC-Task 1 SAF/Axes/Axis 14 - SPARE 1
//     PlcTask Inputs/Main.M14.Axis.NcToPlc <-> Outputs/ToPlc
//     PlcTask Outputs/Main.M14.Axis.PlcToNc <-> Inputs/FromPlc
//   PLC_CRIX_MOT Instance <-> NC-Task 1 SAF/Axes/Axis 15 - SPARE 2
//     PlcTask Inputs/Main.M15.Axis.NcToPlc <-> Outputs/ToPlc
//     PlcTask Outputs/Main.M15.Axis.PlcToNc <-> Inputs/FromPlc
//   PLC_CRIX_MOT Instance <-> NC-Task 1 SAF/Axes/Axis 16 - SDS Injector X
//     PlcTask Inputs/Main.M16.Axis.NcToPlc <-> Outputs/ToPlc
//     PlcTask Outputs/Main.M16.Axis.PlcToNc <-> Inputs/FromPlc
//   PLC_CRIX_MOT Instance <-> NC-Task 1 SAF/Axes/Axis 17 - SDS Injectory Y
//     PlcTask Inputs/Main.M17.Axis.NcToPlc <-> Outputs/ToPlc
//     PlcTask Outputs/Main.M17.Axis.PlcToNc <-> Inputs/FromPlc
//   PLC_CRIX_MOT Instance <-> NC-Task 1 SAF/Axes/Axis 18 - SDS Injector Z
//     PlcTask Inputs/Main.M18.Axis.NcToPlc <-> Outputs/ToPlc
//     PlcTask Outputs/Main.M18.Axis.PlcToNc <-> Inputs/FromPlc
//   PLC_CRIX_MOT Instance <-> NC-Task 1 SAF/Axes/Axis 19 - SDS Rotation X
//     PlcTask Inputs/Main.M19.Axis.NcToPlc <-> Outputs/ToPlc
//     PlcTask Outputs/Main.M19.Axis.PlcToNc <-> Inputs/FromPlc
//   PLC_CRIX_MOT Instance <-> NC-Task 1 SAF/Axes/Axis 2 - Diagnostic Paddle Y
//     PlcTask Inputs/Main.M2.Axis.NcToPlc <-> Outputs/ToPlc
//     PlcTask Outputs/Main.M2.Axis.PlcToNc <-> Inputs/FromPlc
//   PLC_CRIX_MOT Instance <-> NC-Task 1 SAF/Axes/Axis 20 - SDS Jet Rotation
//     PlcTask Inputs/Main.M20.Axis.NcToPlc <-> Outputs/ToPlc
//     PlcTask Outputs/Main.M20.Axis.PlcToNc <-> Inputs/FromPlc
//   PLC_CRIX_MOT Instance <-> NC-Task 1 SAF/Axes/Axis 3 - Diagnostic Paddle Z
//     PlcTask Inputs/Main.M3.Axis.NcToPlc <-> Outputs/ToPlc
//     PlcTask Outputs/Main.M3.Axis.PlcToNc <-> Inputs/FromPlc
//   PLC_CRIX_MOT Instance <-> NC-Task 1 SAF/Axes/Axis 35 - Outcoupling Lens Y
//     PlcTask Inputs/Main.M35.Axis.NcToPlc <-> Outputs/ToPlc
//     PlcTask Outputs/Main.M35.Axis.PlcToNc <-> Inputs/FromPlc
//   PLC_CRIX_MOT Instance <-> NC-Task 1 SAF/Axes/Axis 36 - SDS Z Encoder
//     PlcTask Inputs/Main.M36.Axis.NcToPlc <-> Outputs/ToPlc
//     PlcTask Outputs/Main.M36.Axis.PlcToNc <-> Inputs/FromPlc
//   PLC_CRIX_MOT Instance <-> NC-Task 1 SAF/Axes/Axis 4 - Objectives X
//     PlcTask Inputs/Main.M4.Axis.NcToPlc <-> Outputs/ToPlc
//     PlcTask Outputs/Main.M4.Axis.PlcToNc <-> Inputs/FromPlc
//   PLC_CRIX_MOT Instance <-> NC-Task 1 SAF/Axes/Axis 5 - Objectives Y
//     PlcTask Inputs/Main.M5.Axis.NcToPlc <-> Outputs/ToPlc
//     PlcTask Outputs/Main.M5.Axis.PlcToNc <-> Inputs/FromPlc
//   PLC_CRIX_MOT Instance <-> NC-Task 1 SAF/Axes/Axis 6 - Objectives Z
//     PlcTask Inputs/Main.M6.Axis.NcToPlc <-> Outputs/ToPlc
//     PlcTask Outputs/Main.M6.Axis.PlcToNc <-> Inputs/FromPlc
//   PLC_CRIX_MOT Instance <-> NC-Task 1 SAF/Axes/Axis 7 - Point Detector Y
//     PlcTask Inputs/Main.M7.Axis.NcToPlc <-> Outputs/ToPlc
//     PlcTask Outputs/Main.M7.Axis.PlcToNc <-> Inputs/FromPlc
//   PLC_CRIX_MOT Instance <-> NC-Task 1 SAF/Axes/Axis 8 - Point Detector Rotation
//     PlcTask Inputs/Main.M8.Axis.NcToPlc <-> Outputs/ToPlc
//     PlcTask Outputs/Main.M8.Axis.PlcToNc <-> Inputs/FromPlc
//   PLC_CRIX_MOT Instance <-> NC-Task 1 SAF/Axes/Axis 9 - Illumination X
//     PlcTask Inputs/Main.M9.Axis.NcToPlc <-> Outputs/ToPlc
//     PlcTask Outputs/Main.M9.Axis.PlcToNc <-> Inputs/FromPlc
//   PLC_CRIX_MOT Instance <-> NC-Task 1 SAF/Axes/Camera X
//     PlcTask Inputs/Main.M33.Axis.NcToPlc <-> Outputs/ToPlc
//     PlcTask Outputs/Main.M33.Axis.PlcToNc <-> Inputs/FromPlc
//   PLC_CRIX_MOT Instance <-> NC-Task 1 SAF/Axes/Camera Y
//     PlcTask Inputs/Main.M34.Axis.NcToPlc <-> Outputs/ToPlc
//     PlcTask Outputs/Main.M34.Axis.PlcToNc <-> Inputs/FromPlc
//   PLC_CRIX_MOT Instance <-> NC-Task 1 SAF/Axes/Cryo X
//     PlcTask Inputs/Main.M22.Axis.NcToPlc <-> Outputs/ToPlc
//     PlcTask Outputs/Main.M22.Axis.PlcToNc <-> Inputs/FromPlc
//   PLC_CRIX_MOT Instance <-> NC-Task 1 SAF/Axes/Cryo Y
//     PlcTask Inputs/Main.M23.Axis.NcToPlc <-> Outputs/ToPlc
//     PlcTask Outputs/Main.M23.Axis.PlcToNc <-> Inputs/FromPlc
//   PLC_CRIX_MOT Instance <-> NC-Task 1 SAF/Axes/Cryo Z
//     PlcTask Inputs/Main.M24.Axis.NcToPlc <-> Outputs/ToPlc
//     PlcTask Outputs/Main.M24.Axis.PlcToNc <-> Inputs/FromPlc
//   PLC_CRIX_MOT Instance <-> NC-Task 1 SAF/Axes/Cryo rY
//     PlcTask Inputs/Main.M25.Axis.NcToPlc <-> Outputs/ToPlc
//     PlcTask Outputs/Main.M25.Axis.PlcToNc <-> Inputs/FromPlc
//   PLC_CRIX_MOT Instance <-> NC-Task 1 SAF/Axes/FZP X
//     PlcTask Inputs/Main.M31.Axis.NcToPlc <-> Outputs/ToPlc
//     PlcTask Outputs/Main.M31.Axis.PlcToNc <-> Inputs/FromPlc
//   PLC_CRIX_MOT Instance <-> NC-Task 1 SAF/Axes/FZP Y
//     PlcTask Inputs/Main.M30.Axis.NcToPlc <-> Outputs/ToPlc
//     PlcTask Outputs/Main.M30.Axis.PlcToNc <-> Inputs/FromPlc
//   PLC_CRIX_MOT Instance <-> NC-Task 1 SAF/Axes/FZP Z
//     PlcTask Inputs/Main.M32.Axis.NcToPlc <-> Outputs/ToPlc
//     PlcTask Outputs/Main.M32.Axis.PlcToNc <-> Inputs/FromPlc
//   PLC_CRIX_MOT Instance <-> NC-Task 1 SAF/Axes/M37-X
//     PlcTask Inputs/Main.M37.Axis.NcToPlc <-> Outputs/ToPlc
//     PlcTask Outputs/Main.M37.Axis.PlcToNc <-> Inputs/FromPlc
//   PLC_CRIX_MOT Instance <-> NC-Task 1 SAF/Axes/M38-Y
//     PlcTask Inputs/Main.M38.Axis.NcToPlc <-> Outputs/ToPlc
//     PlcTask Outputs/Main.M38.Axis.PlcToNc <-> Inputs/FromPlc
//   PLC_CRIX_MOT Instance <-> NC-Task 1 SAF/Axes/M39-Z
//     PlcTask Inputs/Main.M39.Axis.NcToPlc <-> Outputs/ToPlc
//     PlcTask Outputs/Main.M39.Axis.PlcToNc <-> Inputs/FromPlc
//   PLC_CRIX_MOT Instance <-> NC-Task 1 SAF/Axes/M40-VLS-Slit-Top
//     PlcTask Inputs/Main.M40.Axis.NcToPlc <-> Outputs/ToPlc
//     PlcTask Outputs/Main.M40.Axis.PlcToNc <-> Inputs/FromPlc
//   PLC_CRIX_MOT Instance <-> NC-Task 1 SAF/Axes/M41-VLS-Slit-Bottom
//     PlcTask Inputs/Main.M41.Axis.NcToPlc <-> Outputs/ToPlc
//     PlcTask Outputs/Main.M41.Axis.PlcToNc <-> Inputs/FromPlc
//   PLC_CRIX_MOT Instance <-> NC-Task 1 SAF/Axes/M42-VLS-Slit-Right
//     PlcTask Inputs/Main.M42.Axis.NcToPlc <-> Outputs/ToPlc
//     PlcTask Outputs/Main.M42.Axis.PlcToNc <-> Inputs/FromPlc
//   PLC_CRIX_MOT Instance <-> NC-Task 1 SAF/Axes/M43-VLS-Slit-Left
//     PlcTask Inputs/Main.M43.Axis.NcToPlc <-> Outputs/ToPlc
//     PlcTask Outputs/Main.M43.Axis.PlcToNc <-> Inputs/FromPlc
//   PLC_CRIX_MOT Instance <-> NC-Task 1 SAF/Axes/M44-VLS-Mirror-Pitch
//     PlcTask Inputs/Main.M44.Axis.NcToPlc <-> Outputs/ToPlc
//     PlcTask Outputs/Main.M44.Axis.PlcToNc <-> Inputs/FromPlc
//   PLC_CRIX_MOT Instance <-> NC-Task 1 SAF/Axes/M45-VLS-Grating-Pitch
//     PlcTask Inputs/Main.M45.Axis.NcToPlc <-> Outputs/ToPlc
//     PlcTask Outputs/Main.M45.Axis.PlcToNc <-> Inputs/FromPlc
//   PLC_CRIX_MOT Instance <-> NC-Task 1 SAF/Axes/M46-VLS-Camera-Pitch
//     PlcTask Inputs/Main.M46.Axis.NcToPlc <-> Outputs/ToPlc
//     PlcTask Outputs/Main.M46.Axis.PlcToNc <-> Inputs/FromPlc
//   PLC_CRIX_MOT Instance <-> NC-Task 1 SAF/Axes/M47-VLS-Camera-Dist
//     PlcTask Inputs/Main.M47.Axis.NcToPlc <-> Outputs/ToPlc
//     PlcTask Outputs/Main.M47.Axis.PlcToNc <-> Inputs/FromPlc
//   PLC_CRIX_MOT Instance <-> NC-Task 1 SAF/Axes/M48- Cryopump Y10
//     PlcTask Inputs/Main.M48.Axis.NcToPlc <-> Outputs/ToPlc
//     PlcTask Outputs/Main.M48.Axis.PlcToNc <-> Inputs/FromPlc
//   PLC_CRIX_MOT Instance <-> NC-Task 1 SAF/Axes/M49- Cryopump Y11
//     PlcTask Inputs/Main.M49.Axis.NcToPlc <-> Outputs/ToPlc
//     PlcTask Outputs/Main.M49.Axis.PlcToNc <-> Inputs/FromPlc
//   PLC_CRIX_MOT Instance <-> NC-Task 1 SAF/Axes/RCI RX
//     PlcTask Inputs/Main.M29.Axis.NcToPlc <-> Outputs/ToPlc
//     PlcTask Outputs/Main.M29.Axis.PlcToNc <-> Inputs/FromPlc
//   PLC_CRIX_MOT Instance <-> NC-Task 1 SAF/Axes/RCI X
//     PlcTask Inputs/Main.M26.Axis.NcToPlc <-> Outputs/ToPlc
//     PlcTask Outputs/Main.M26.Axis.PlcToNc <-> Inputs/FromPlc
//   PLC_CRIX_MOT Instance <-> NC-Task 1 SAF/Axes/RCI Y
//     PlcTask Inputs/Main.M27.Axis.NcToPlc <-> Outputs/ToPlc
//     PlcTask Outputs/Main.M27.Axis.PlcToNc <-> Inputs/FromPlc
//   PLC_CRIX_MOT Instance <-> NC-Task 1 SAF/Axes/RCI Z
//     PlcTask Inputs/Main.M28.Axis.NcToPlc <-> Outputs/ToPlc
//     PlcTask Outputs/Main.M28.Axis.PlcToNc <-> Inputs/FromPlc
//   PLC_CRIX_MOT Instance <-> NC-Task 1 SAF/Axes/SL2K2-BOTTOM-M50
//     PlcTask Inputs/Main.M50.Axis.NcToPlc <-> Outputs/ToPlc
//     PlcTask Outputs/Main.M50.Axis.PlcToNc <-> Inputs/FromPlc
//   PLC_CRIX_MOT Instance <-> NC-Task 1 SAF/Axes/SL2K2-NORTH-M52
//     PlcTask Inputs/Main.M52.Axis.NcToPlc <-> Outputs/ToPlc
//     PlcTask Outputs/Main.M52.Axis.PlcToNc <-> Inputs/FromPlc
//   PLC_CRIX_MOT Instance <-> NC-Task 1 SAF/Axes/SL2K2-SOUTH-M53
//     PlcTask Inputs/Main.M53.Axis.NcToPlc <-> Outputs/ToPlc
//     PlcTask Outputs/Main.M53.Axis.PlcToNc <-> Inputs/FromPlc
//   PLC_CRIX_MOT Instance <-> NC-Task 1 SAF/Axes/SL2K2-TOP-M51
//     PlcTask Inputs/Main.M51.Axis.NcToPlc <-> Outputs/ToPlc
//     PlcTask Outputs/Main.M51.Axis.PlcToNc <-> Inputs/FromPlc

// ---- DUTs/EPS/ST_EPSLimits.TcDUT
TYPE ST_EPSLimits :
    // Defines the PLC limits and EPS structure where these limits are valid
STRUCT
    {attribute 'pytmc' := 'pv: FwdLimit'}
    // Forward Limit
    fFwd_Limits : LREAL;
    {attribute 'pytmc' := 'pv: BwdLimit'}
    // Backward Limit
    fBwd_Limits	: LREAL;
    {attribute 'pytmc' := 'pv: ST'}
    // EPS_OK - TRUE, Use limits as 'plc limits'; EPS_OK - FALSE, DO not use limits
    stEPS 		: DUT_EPS;
END_STRUCT
END_TYPE

// ---- GVLs/GVL_FiberLite.TcGVL
//{attribute 'qualified_only'}
VAR_GLOBAL
    //Fiber-Lite Control
    {attribute 'TcLinkTo' := '.iIlluminatorINT := TIID^Device 1 (EtherCAT)^Term 5 (EK1200)^Term 6 (EK1122-0080)^DRL02-EK0 (EK1101-0080)^DRL02-ECJ1 (EK1122)^CryoStat (EK1101)^Term 158 (EL4004)^AO Outputs Channel 1^Analog output'}
    {attribute 'pytmc' := '
        pv: RIX:CRIX:LED:01
        io: io
    '}

    bLedOutput1 : FB_LED;

    {attribute 'TcLinkTo' := '.iIlluminatorINT := TIID^Device 1 (EtherCAT)^Term 5 (EK1200)^Term 6 (EK1122-0080)^DRL02-EK0 (EK1101-0080)^DRL02-ECJ1 (EK1122)^CryoStat (EK1101)^FiberLite (EL4004)^AO Outputs Channel 2^Analog output'}
    {attribute 'pytmc' := '
        pv: RIX:CRIX:LED:02
        io: io
    '}

    bLedOutput2 : FB_LED;

       {attribute 'TcLinkTo' := '.iIlluminatorINT := TIID^Device 1 (EtherCAT)^Term 5 (EK1200)^Term 6 (EK1122-0080)^DRL02-EK0 (EK1101-0080)^DRL02-ECJ1 (EK1122)^CryoStat (EK1101)^FiberLite (EL4004)^AO Outputs Channel 3^Analog output'}
    {attribute 'pytmc' := '
        pv: RIX:CRIX:LED:03
        io: io
    '}

    bLedOutput3 : FB_LED;

       {attribute 'TcLinkTo' := '.iIlluminatorINT := TIID^Device 1 (EtherCAT)^Term 5 (EK1200)^Term 6 (EK1122-0080)^DRL02-EK0 (EK1101-0080)^DRL02-ECJ1 (EK1122)^CryoStat (EK1101)^FiberLite (EL4004)^AO Outputs Channel 4^Analog output'}
    {attribute 'pytmc' := '
        pv: RIX:CRIX:LED:04
        io: io
    '}

    bLedOutput4 : FB_LED;

END_VAR

// ---- GVLs/GVL_MotorEPS.TcGVL
VAR_GLOBAL

    fDPL_X  	: LREAL;
    fDPL_Z 		: LREAL;
    fDPL_Y 		: LREAL;

    fSDS_RX 	: LREAL;
    fSDS_Y 		: LREAL;
    fSDS_Z_ENC 	: LREAL;

    fRCC_Z 		: LREAL;
    fRCC_Y 		: LREAL;

    fOBJ_X		: LREAL;

    tEPS_OVRD_RESET_TIME : TIME := T#5m; // Resets overide after this amount of time.


     {attribute 'pytmc' := '
        pv: RIX:CRIX:EPS:fNozzleCatcherOffset
        io: io
    '}
    fNozzleCatcherOffset	: LREAL := 20;

END_VAR

// ---- GVLs/Main.TcGVL
	//{attribute 'qualified_only'}
VAR_GLOBAL

